ABB RobotStudio station: IRB1600_packaged.rspag

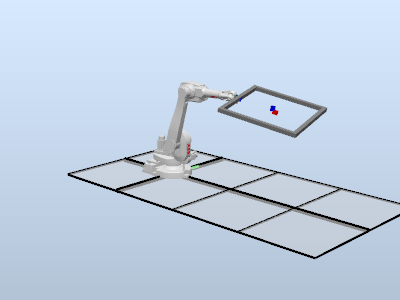
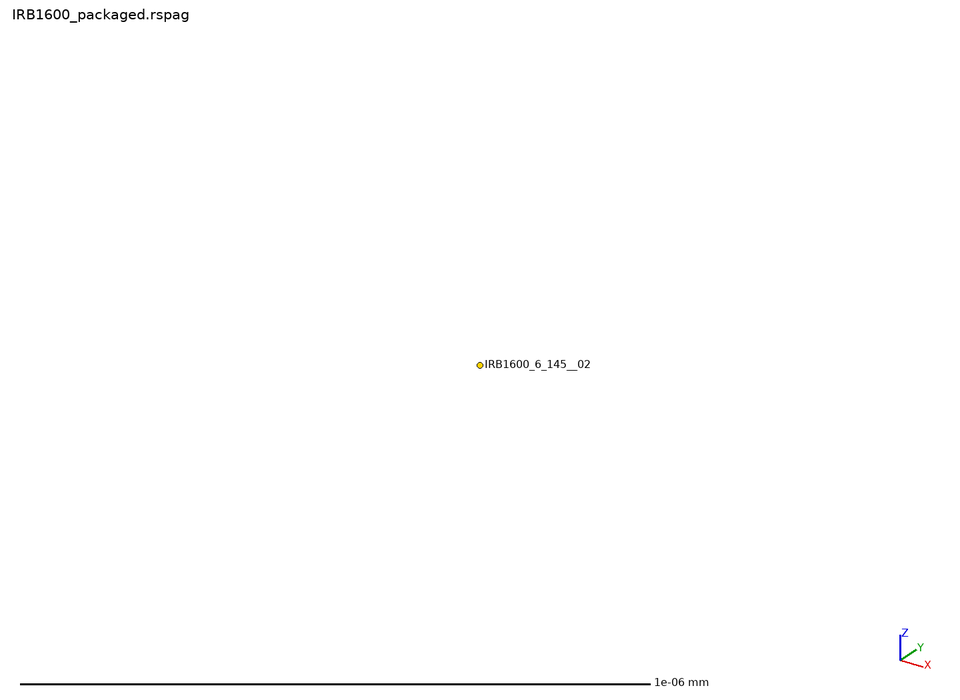
[picture v1: parts stored in the station drawn from their meshes, with robot base, taught points and paths (robot models come from the ABB library and are not in the file)]
--- station ---
Station Solution1 (saved by RobotStudio 22.2.9947.0)
Controller IRB1600_6_145
  mechanical unit ROB_1: IRB1600_6_145__02, 6 joints, base frame (0, 0, 0) mm
Layout (positions relative to the parent item):
  - IRB1600_6_145__02 [mechanism, from Robots\IRB1600_6_145_G_02.rslib] at (0, 0, 0) mm; joint values [0.1292, 0.2457, -0.2431, -2.5339, -0.2406, 2.6375] (rad or m)
  - flange_connector [part, from Tools\IsoPlate_small_Binzel.rslib] at (974.03, 135.42, 1151.03) mm, rotated rx 149.84 ry 76.75 rz 164.54 deg
  - plane [part] at (1455.82, 269.91, 1054.92) mm, rotated rx 173.25 ry -11.43 rz -164.62 deg, size 1000 x 1000 x 50 mm
  - Frame_1 [frame]
  - Frame_2 [frame] at (-23.65, -1.83, 250.36) mm
Attachment: flange_connector is attached to IRB1600_6_145__02 / Link6
Attachment: plane is attached to flange_connector
Attachment: Workobject_2 is attached to IRB1600_6_145__02 / Link1
Targets, tools, work objects and paths stored in the station and not in the controller backup, written as RAPID:
! task T_ROB1
MODULE Module1
  LOCAL PERS wobjdata egm_wobj:=[FALSE,TRUE,"",[[0,0,0],[1,0,0,0]],[[0,0,0],[1,0,0,0]]];
  PROC EGM_CARTESIAN_MOVE()
    WaitTime 2;
  ENDPROC
ENDMODULE


--- Backups/IRB1600_6_145/RAPID/TASK1/PROGMOD/CalibData.mod ---
MODULE CalibData
    TASK PERS tooldata Tooldata_3:=[TRUE,[[-23.481,11.123,47.179],[0.707106781,0,0.707106781,0]],[1,[0,0,1],[1,0,0,0],0,0,0]];
    TASK PERS tooldata Tooldata_8:=[TRUE,[[35.292999999,18.761,1471.373000001],[0.707106781,0,-0.707106781,0]],[1,[0,0,1],[1,0,0,0],0,0,0]];
    TASK PERS tooldata Tooldata_4:=[TRUE,[[0,0,0],[1,0,0,0]],[1,[0,0,1],[1,0,0,0],0,0,0]];
    TASK PERS tooldata Tooldata_5:=[TRUE,[[0,0,0],[1,0,0,0]],[1,[0,0,1],[1,0,0,0],0,0,0]];
    TASK PERS tooldata Tooldata_6:=[TRUE,[[0,0,0],[1,0,0,0]],[1,[0,0,1],[1,0,0,0],0,0,0]];
    TASK PERS tooldata Tooldata_7:=[TRUE,[[-23.772999698,2.161000196,740.120999999],[0.707106781,0,-0.707106781,0]],[1,[0,0,1],[1,0,0,0],0,0,0]];
    TASK PERS wobjdata Workobject_2:=[FALSE,TRUE,"ROB_1",[[-55.133477186,-6.202200727,258.13059393],[1,0,0,0]],[[0,0,0],[1,0,0,0]]];
    TASK PERS tooldata Tooldata_9:=[TRUE,[[20.616002648,0.899999913,497.265999882],[0.707106781,-0.000000002,-0.707106781,0]],[1,[0,0,1],[1,0,0,0],0,0,0]];
    TASK PERS wobjdata Wobj_joint1:=[TRUE,FALSE,"ROB_1",[[639.116,-613.962,-938.233],[1,0,0,0]],[[0,0,0],[1,0,0,0]]];
ENDMODULE

--- Backups/IRB1600_6_145/RAPID/TASK1/PROGMOD/Module1.mod ---
MODULE Module1

     VAR robtarget position;
     VAR robtarget starting_position;
     VAR jointtarget joints;
     VAR speeddata velocity;
    TASK PERS wobjdata wobj:=[FALSE,FALSE,"ROB_1",[[639.116,-22.796,-980.437],[1,0,0,0]],[[0,0,0],[1,0,0,0]]];

    PROC main()

starting_position := CRobT(\TaskName:="T_ROB1" \Tool:=Tooldata_9 \WObj:=Workobject_2);
move 64,-487.9,0,3.2,0,1.3;
move 64,-487.9,0,3.2,15,1.4;
move 64,-487.9,0,3.6,15,1.4;
move 65,-487.9,-0,3.6,15,1.4;
move 65,-487.9,-0,3.6,15,1.5;
move 65,-487.9,-0.1,3.6,15,1.5;
move 65,-487.9,-0.1,3.6,15,1.6;
move 65,-487.9,-0.1,3.6,15,1.6;
move 66,-488,-0.1,3.6,15,1.7;
move 66,-488.1,-0.2,3.6,14.9,1.7;
move 66,-488.1,-0.2,3.6,14.9,1.8;
move 66,-488.2,-0.2,3.6,14.9,1.9;
move 66,-488.3,-0.2,3.6,14.9,1.9;
move 66,-488.5,-0.3,3.6,14.9,2;
move 66,-488.6,-0.3,3.6,14.9,2.1;
move 66,-488.8,-0.3,3.6,14.8,2.1;
move 66,-489,-0.3,3.6,14.8,2.2;
move 66,-489.3,-0.4,3.6,14.8,2.3;
move 66,-489.6,-0.4,3.6,14.8,2.3;
move 66,-489.9,-0.4,3.6,14.8,2.4;
move 66,-490.4,-0.5,3.6,14.7,2.5;
move 66,-490.8,-0.5,3.6,14.7,2.5;
move 66,-491.3,-0.5,3.6,14.7,2.6;
move 66,-491.9,-0.6,3.6,14.6,2.7;
move 66,-492.5,-0.6,3.6,14.6,2.8;
move 66,-493.2,-0.6,3.6,14.6,2.9;
move 65,-493.9,-0.7,3.6,14.5,2.9;
move 65,-494.7,-0.7,3.6,14.5,3;
move 65,-495.5,-0.7,3.6,14.5,3.1;
move 65,-496.4,-0.8,3.6,14.4,3.2;
move 64,-497.4,-0.8,3.6,14.4,3.3;
move 64,-498.4,-0.8,3.6,14.3,3.4;
move 63,-499.4,-0.9,3.6,14.3,3.5;
move 62,-500.5,-0.9,3.2,14.2,3.6;
move 62,-501.6,-0.9,3.2,14.2,3.7;
move 61,-502.7,-1,3.2,14.1,3.8;
move 60,-503.8,-1,3.2,14.1,3.8;
move 60,-504.9,-1,3.2,14,3.9;
move 59,-506,-1.1,3.2,14,4;
move 58,-507.1,-1.1,3.2,13.9,4.1;
move 57,-508.2,-1.1,3.2,13.9,4.2;
move 56,-509.2,-1.2,2.8,13.8,4.3;
move 55,-510.3,-1.2,2.8,13.8,4.4;
move 54,-511.3,-1.2,2.8,13.7,4.5;
move 53,-512.3,-1.3,2.8,13.6,4.6;
move 52,-513.2,-1.3,2.8,13.6,4.7;
move 51,-514,-1.3,2.4,13.5,4.8;
move 50,-514.8,-1.3,2.4,13.5,4.9;
move 49,-515.5,-1.4,2.4,13.4,5;
move 47,-516.2,-1.4,2.4,13.3,5.1;
move 46,-516.8,-1.4,2.4,13.3,5.2;
move 45,-517.3,-1.4,2,13.2,5.3;
move 44,-517.7,-1.4,2,13.1,5.4;
move 42,-518.1,-1.4,2,13,5.5;
move 41,-518.3,-1.5,2,13,5.6;
move 39,-518.5,-1.5,1.6,12.9,5.7;
move 38,-518.6,-1.5,1.6,12.8,5.8;
move 37,-518.6,-1.5,1.6,12.7,5.9;
move 35,-518.5,-1.5,1.6,12.7,6;
move 34,-518.3,-1.5,1.2,12.6,6.1;
move 32,-518.1,-1.5,1.2,12.5,6.2;
move 31,-517.8,-1.5,1.2,12.4,6.2;
move 30,-517.5,-1.6,1.2,12.3,6.3;
move 28,-517.2,-1.6,0.8,12.3,6.4;
move 27,-516.8,-1.6,0.8,12.2,6.5;
move 25,-516.4,-1.6,0.8,12.1,6.6;
move 24,-516.1,-1.6,0.8,12,6.7;
move 22,-515.7,-1.5,0.4,11.9,6.8;
move 21,-515.3,-1.5,0.4,11.8,6.9;
move 20,-515,-1.5,0.4,11.7,7;
move 18,-514.6,-1.5,0.4,11.6,7;
move 17,-514.3,-1.5,0,11.6,7.1;
move 15,-514.1,-1.5,0,11.5,7.2;
move 14,-513.8,-1.5,-0,11.4,7.3;
move 13,-513.7,-1.5,-0,11.3,7.4;
move 12,-513.5,-1.5,-0.4,11.2,7.5;
move 10,-513.4,-1.5,-0.4,11.1,7.5;
move 9,-513.3,-1.4,-0.4,11,7.6;
move 8,-513.2,-1.4,-0.4,10.9,7.7;
move 7,-513.2,-1.4,-0.4,10.8,7.8;
move 6,-513.2,-1.4,-0.8,10.7,7.9;
move 4,-513.2,-1.4,-0.8,10.6,7.9;
move 3,-513.2,-1.3,-0.8,10.5,8;
move 2,-513.1,-1.3,-0.8,10.4,8.1;
move 1,-513.1,-1.3,-0.8,10.3,8.2;
move 0,-513.1,-1.3,-1.2,10.2,8.2;
move -1,-513.1,-1.3,-1.2,10.1,8.3;
move -2,-513,-1.2,-1.2,9.9,8.4;
move -3,-513,-1.2,-1.2,9.8,8.4;
move -4,-512.9,-1.2,-1.2,9.7,8.5;
move -5,-512.8,-1.2,-1.2,9.6,8.6;
move -5,-512.7,-1.2,-1.6,9.5,8.7;
move -6,-512.5,-1.1,-1.6,9.4,8.7;
move -7,-512.3,-1.1,-1.6,9.3,8.8;
move -7,-512,-1.1,-1.6,9.2,8.9;
move -7,-511.7,-1.1,-1.6,9,8.9;
move -8,-511.4,-1,-1.6,8.9,9;
move -8,-511,-1,-1.6,8.8,9.1;
move -8,-510.6,-1,-1.6,8.7,9.1;
move -8,-510.2,-1,-1.6,8.6,9.2;
move -8,-509.7,-1,-1.6,8.5,9.3;
move -8,-509.1,-1,-1.6,8.3,9.3;
move -8,-508.6,-0.9,-1.6,8.2,9.4;
move -8,-508,-0.9,-1.6,8.1,9.4;
move -9,-507.4,-0.9,-1.6,8,9.5;
move -9,-506.8,-0.9,-1.6,7.9,9.6;
move -9,-506.2,-0.9,-1.6,7.7,9.6;
move -9,-505.6,-0.9,-2,7.6,9.7;
move -9,-505,-0.9,-1.6,7.5,9.7;
move -9,-504.4,-0.8,-1.6,7.4,9.8;
move -9,-503.8,-0.8,-1.6,7.2,9.8;
move -8,-503.2,-0.8,-1.6,7.1,9.9;
move -8,-502.7,-0.8,-1.6,7,9.9;
move -8,-502.2,-0.8,-1.6,6.9,10;
move -8,-501.7,-0.8,-1.6,6.7,10;
move -8,-501.2,-0.8,-1.6,6.6,10.1;
move -8,-500.8,-0.8,-1.6,6.5,10.1;
move -7,-500.4,-0.7,-1.6,6.4,10.2;
move -7,-500,-0.7,-1.6,6.2,10.2;
move -7,-499.7,-0.7,-1.6,6.1,10.3;
move -6,-499.4,-0.7,-1.6,6,10.3;
move -6,-499.1,-0.7,-1.6,5.8,10.4;
move -5,-498.8,-0.7,-1.2,5.7,10.4;
move -4,-498.6,-0.7,-1.2,5.6,10.4;
move -4,-498.3,-0.7,-1.2,5.5,10.5;
move -3,-498.1,-0.7,-1.2,5.3,10.5;
move -2,-497.9,-0.7,-1.2,5.2,10.5;
move -1,-497.7,-0.7,-1.2,5.1,10.6;
move -1,-497.5,-0.6,-1.2,4.9,10.6;
move 0,-497.3,-0.6,-1.2,4.8,10.6;
move 1,-497.1,-0.6,-0.8,4.7,10.7;
move 2,-496.9,-0.6,-0.8,4.5,10.7;
move 3,-496.8,-0.6,-0.8,4.4,10.7;
move 4,-496.6,-0.6,-0.8,4.3,10.7;
move 5,-496.5,-0.6,-0.8,4.1,10.8;
move 6,-496.4,-0.6,-0.8,4,10.8;
move 7,-496.3,-0.6,-0.4,3.9,10.8;
move 7,-496.1,-0.6,-0.4,3.7,10.8;
move 8,-496,-0.6,-0.4,3.6,10.8;
move 9,-495.9,-0.6,-0.4,3.5,10.9;
move 10,-495.8,-0.6,-0.4,3.3,10.9;
move 11,-495.8,-0.6,-0.4,3.2,10.9;
move 12,-495.7,-0.6,-0,3,10.9;
move 12,-495.6,-0.5,-0,2.9,10.9;
move 13,-495.6,-0.5,-0,2.8,10.9;
move 14,-495.5,-0.5,-0,2.6,10.9;
move 14,-495.5,-0.5,0,2.5,10.9;
move 14,-495.5,-0.5,0,2.4,10.9;
move 15,-495.6,-0.5,0,2.2,11;
move 15,-495.6,-0.5,0,2.1,11;
move 16,-495.7,-0.5,0,2,11;
move 16,-495.8,-0.5,0,1.8,11;
move 17,-495.9,-0.5,0,1.7,11;
move 17,-496,-0.5,0,1.6,11;
move 18,-496.2,-0.5,0.4,1.4,11;
move 18,-496.4,-0.5,0.4,1.3,11;
move 19,-496.6,-0.4,0.4,1.1,11;
move 19,-496.8,-0.4,0.4,1,11;
move 20,-497.1,-0.4,0.4,0.9,11;
move 20,-497.4,-0.4,0.4,0.7,11;
move 20,-497.8,-0.4,0.4,0.6,11;
move 20,-498.2,-0.4,0.4,0.5,11;
move 20,-498.6,-0.4,0.4,0.3,11;
move 19,-499.1,-0.4,0.4,0.2,11;
move 19,-499.6,-0.4,0.4,0.1,11;
move 18,-500.1,-0.4,0.4,-0.1,11;
move 18,-500.7,-0.4,0.4,-0.2,11;
move 17,-501.2,-0.4,0,-0.3,11;
move 16,-501.8,-0.4,0,-0.5,11;
move 16,-502.4,-0.3,0,-0.6,11;
move 15,-503,-0.3,0,-0.7,11;
move 15,-503.6,-0.3,0,-0.9,11;
move 14,-504.3,-0.3,-0,-1,11;
move 13,-504.8,-0.3,-0,-1.1,11;
move 13,-505.4,-0.3,-0,-1.3,11;
move 12,-506,-0.3,-0,-1.4,11;
move 11,-506.5,-0.3,-0.4,-1.5,11;
move 10,-506.9,-0.3,-0.4,-1.7,11;
move 9,-507.3,-0.3,-0.4,-1.8,11;
move 8,-507.7,-0.3,-0.4,-1.9,11;
move 7,-508,-0.3,-0.4,-2,11;
move 6,-508.3,-0.3,-0.4,-2.2,11;
move 5,-508.5,-0.3,-0.8,-2.3,11;
move 4,-508.6,-0.3,-0.8,-2.4,11;
move 3,-508.7,-0.3,-0.8,-2.6,11;
move 2,-508.8,-0.3,-0.8,-2.7,11;
move 1,-508.7,-0.3,-0.8,-2.8,10.9;
move -1,-508.6,-0.3,-1.2,-2.9,10.9;
move -2,-508.5,-0.3,-1.2,-3.1,10.9;
move -3,-508.3,-0.2,-1.2,-3.2,10.9;
move -5,-508,-0.2,-1.2,-3.3,10.9;
move -6,-507.7,-0.2,-1.6,-3.4,10.9;
move -7,-507.3,-0.2,-1.6,-3.6,10.9;
move -9,-506.9,-0.2,-1.6,-3.7,10.9;
move -10,-506.5,-0.2,-1.6,-3.8,10.8;
move -11,-506,-0.2,-2,-3.9,10.8;
move -12,-505.4,-0.2,-2,-4,10.8;
move -14,-504.9,-0.2,-2,-4.2,10.8;
move -15,-504.3,-0.2,-2,-4.3,10.8;
move -16,-503.7,-0.2,-2,-4.4,10.7;
move -17,-503.1,-0.2,-2.4,-4.5,10.7;
move -18,-502.5,-0.2,-2.4,-4.6,10.7;
move -19,-501.8,-0.1,-2.4,-4.8,10.7;
move -20,-501.2,-0.1,-2.4,-4.9,10.6;
move -21,-500.6,-0.1,-2.4,-5,10.6;
move -22,-500,-0.1,-2.8,-5.1,10.6;
move -23,-499.4,-0.1,-2.8,-5.2,10.6;
move -24,-498.8,-0.1,-2.8,-5.3,10.5;
move -25,-498.2,-0.1,-2.8,-5.5,10.5;
move -26,-497.6,-0.1,-2.8,-5.6,10.5;
move -27,-497.1,-0,-2.8,-5.7,10.4;
move -27,-496.6,0,-2.8,-5.8,10.4;
move -28,-496,0,-3.2,-5.9,10.3;
move -29,-495.5,0,-3.2,-6,10.3;
move -30,-495,0,-3.2,-6.1,10.3;
move -30,-494.5,0.1,-3.2,-6.2,10.2;
move -31,-493.9,0.1,-3.2,-6.3,10.2;
move -31,-493.4,0.1,-3.2,-6.4,10.1;
move -32,-492.8,0.2,-3.2,-6.5,10.1;
move -32,-492.2,0.2,-3.2,-6.6,10;
move -32,-491.7,0.2,-3.6,-6.7,10;
move -33,-491.1,0.3,-3.2,-6.9,9.9;
move -33,-490.4,0.3,-3.2,-7,9.9;
move -33,-489.8,0.3,-3.2,-7.1,9.8;
move -33,-489.2,0.3,-3.6,-7.2,9.8;
move -33,-488.5,0.4,-3.6,-7.3,9.7;
move -33,-487.9,0.4,-3.6,-7.4,9.7;
move -33,-487.3,0.4,-3.6,-7.4,9.6;
move -33,-486.7,0.5,-3.2,-7.5,9.6;
move -32,-486.1,0.5,-3.2,-7.6,9.5;
move -32,-485.5,0.6,-3.2,-7.7,9.5;
move -32,-485,0.6,-3.2,-7.8,9.4;
move -31,-484.4,0.6,-3.2,-7.9,9.4;
move -31,-483.9,0.7,-3.2,-8,9.3;
move -31,-483.4,0.7,-3.2,-8.1,9.2;
move -31,-482.9,0.8,-3.2,-8.2,9.2;
move -30,-482.5,0.8,-3.2,-8.3,9.1;
move -30,-482,0.9,-3.2,-8.4,9.1;
move -29,-481.6,0.9,-3.2,-8.5,9;
move -29,-481.2,0.9,-3.2,-8.5,9;
move -28,-480.8,1,-3.2,-8.6,8.9;
move -27,-480.4,1,-2.8,-8.7,8.8;
move -26,-480,1.1,-2.8,-8.8,8.8;
move -26,-479.5,1.1,-2.8,-8.9,8.7;
move -25,-479.1,1.2,-2.8,-9,8.6;
move -24,-478.6,1.2,-2.8,-9,8.6;
move -23,-478.1,1.3,-2.8,-9.1,8.5;
move -22,-477.6,1.3,-2.4,-9.2,8.5;
move -20,-477.1,1.4,-2.4,-9.3,8.4;
move -19,-476.5,1.4,-2.4,-9.4,8.3;
move -18,-475.9,1.5,-2.4,-9.4,8.3;
move -17,-475.3,1.5,-2.4,-9.5,8.2;
move -16,-474.7,1.6,-2,-9.6,8.1;
move -14,-474.1,1.6,-2,-9.7,8.1;
move -13,-473.4,1.7,-2,-9.7,8;
move -12,-472.7,1.7,-2,-9.8,7.9;
move -10,-472,1.7,-1.6,-9.9,7.9;
move -9,-471.4,1.8,-1.6,-9.9,7.8;
move -8,-470.7,1.8,-1.6,-10,7.7;
move -6,-470,1.9,-1.6,-10.1,7.7;
move -5,-469.4,1.9,-1.2,-10.1,7.6;
move -4,-468.8,1.9,-1.2,-10.2,7.5;
move -3,-468.3,2,-1.2,-10.3,7.4;
move -1,-467.9,2,-1.2,-10.3,7.4;
move 0,-467.5,2.1,-1.2,-10.4,7.3;
move 1,-467.2,2.1,-0.8,-10.4,7.2;
move 3,-467,2.1,-0.8,-10.5,7.1;
move 4,-466.9,2.1,-0.8,-10.5,7.1;
move 5,-466.9,2.2,-0.8,-10.6,7;
move 7,-466.9,2.2,-0.4,-10.7,6.9;
move 8,-467,2.2,-0.4,-10.7,6.9;
move 10,-467.2,2.2,-0.4,-10.8,6.8;
move 11,-467.5,2.3,-0.4,-10.8,6.7;
move 12,-467.9,2.3,-0,-10.9,6.6;
move 14,-468.3,2.3,-0,-10.9,6.5;
move 15,-468.8,2.3,0,-11,6.5;
move 16,-469.4,2.3,0,-11,6.4;
move 17,-470,2.3,0.4,-11.1,6.3;
move 18,-470.7,2.3,0.4,-11.1,6.2;
move 20,-471.4,2.3,0.4,-11.1,6.2;
move 21,-472.1,2.3,0.4,-11.2,6.1;
move 21,-472.8,2.3,0.4,-11.2,6;
move 22,-473.6,2.3,0.4,-11.3,5.9;
move 23,-474.3,2.3,0.8,-11.3,5.8;
move 24,-475.1,2.3,0.8,-11.4,5.8;
move 25,-475.8,2.3,0.8,-11.4,5.7;
move 25,-476.5,2.3,0.8,-11.4,5.6;
move 26,-477.1,2.3,0.8,-11.5,5.5;
move 26,-477.8,2.3,0.8,-11.5,5.4;
move 27,-478.3,2.3,0.8,-11.5,5.4;
move 27,-478.9,2.2,0.8,-11.6,5.3;
move 28,-479.4,2.2,0.8,-11.6,5.2;
move 28,-479.8,2.2,0.8,-11.6,5.1;
move 29,-480.2,2.2,1.2,-11.7,5;
move 30,-480.6,2.1,1.2,-11.7,5;
move 30,-480.9,2.1,1.2,-11.7,4.9;
move 31,-481.2,2.1,1.2,-11.7,4.8;
move 31,-481.5,2.1,1.2,-11.8,4.7;
move 31,-481.7,2,1.2,-11.8,4.6;
move 31,-481.9,2,1.2,-11.8,4.5;
move 31,-482.1,2,1.2,-11.8,4.5;
move 32,-482.2,1.9,1.2,-11.8,4.4;
move 32,-482.4,1.9,1.2,-11.9,4.3;
move 32,-482.5,1.8,1.2,-11.9,4.2;
move 32,-482.6,1.8,1.2,-11.9,4.1;
move 32,-482.7,1.8,1.2,-11.9,4;
move 32,-482.8,1.7,1.2,-11.9,4;
move 32,-482.9,1.7,1.2,-11.9,3.9;
move 32,-483,1.6,1.2,-12,3.8;
move 32,-483.1,1.6,1.2,-12,3.7;
move 32,-483.2,1.5,1.2,-12,3.6;
move 32,-483.2,1.5,1.2,-12,3.5;
move 32,-483.2,1.4,1.2,-12,3.5;
move 32,-483.3,1.4,1.2,-12,3.4;
move 31,-483.3,1.3,1.2,-12,3.3;
move 31,-483.3,1.3,1.2,-12,3.2;
move 31,-483.3,1.2,1.2,-12,3.1;
move 31,-483.3,1.2,1.2,-12,3;
move 30,-483.4,1.1,1.2,-12,2.9;
move 30,-483.4,1.1,1.2,-12,2.9;
move 29,-483.4,1,1.2,-12,2.8;
move 29,-483.5,1,0.8,-12,2.7;
move 28,-483.5,0.9,0.8,-12,2.6;
move 27,-483.5,0.9,0.8,-12,2.5;
move 27,-483.5,0.8,0.8,-12,2.4;
move 27,-483.5,0.8,0.8,-12,2.3;
move 26,-483.5,0.8,0.8,-12,2.3;
move 26,-483.5,0.7,0.8,-12,2.2;
move 26,-483.5,0.7,0.8,-12,2.1;
move 26,-483.5,0.6,0.8,-12,2;
move 26,-483.5,0.6,0.8,-12,1.9;
move 26,-483.5,0.5,0.8,-12,1.8;
move 26,-483.5,0.4,0.8,-12,1.7;
move 26,-483.5,0.4,0.8,-11.9,1.7;
move 26,-483.5,0.3,0.8,-11.9,1.6;
move 27,-483.5,0.3,0.8,-11.9,1.5;
move 27,-483.5,0.3,0.8,-11.9,1.4;
move 27,-483.5,0.2,0.8,-11.9,1.3;
move 28,-483.5,0.1,0.8,-11.9,1.2;
move 28,-483.5,0.1,0.8,-11.9,1.2;
move 29,-483.5,0,1.2,-11.8,1.1;
move 30,-483.5,-0,1.2,-11.8,1;
move 30,-483.5,-0.1,1.2,-11.8,0.9;
move 31,-483.5,-0.1,1.2,-11.8,0.8;
move 31,-483.5,-0.1,1.2,-11.8,0.7;
move 31,-483.5,-0.1,1.2,-11.7,0.7;
move 31,-483.5,-0.2,1.2,-11.7,0.6;
move 31,-483.5,-0.3,1.2,-11.7,0.5;
move 32,-483.5,-0.3,1.2,-11.7,0.4;
move 32,-483.5,-0.3,1.2,-11.6,0.3;
move 32,-483.5,-0.4,1.2,-11.6,0.2;
move 32,-483.5,-0.4,1.2,-11.6,0.2;
move 32,-483.5,-0.5,1.2,-11.5,0.1;
move 33,-483.5,-0.5,1.2,-11.5,-0;
move 33,-483.5,-0.5,1.2,-11.5,-0.1;
move 34,-483.5,-0.6,1.2,-11.5,-0.2;
move 34,-483.5,-0.6,1.2,-11.4,-0.3;
move 35,-483.5,-0.7,1.6,-11.4,-0.3;
move 35,-483.5,-0.7,1.6,-11.4,-0.4;
move 36,-483.5,-0.7,1.6,-11.3,-0.5;
move 36,-483.5,-0.8,1.6,-11.3,-0.6;
move 37,-483.5,-0.8,1.6,-11.3,-0.7;
move 37,-483.5,-0.9,1.6,-11.2,-0.7;
move 38,-483.5,-0.9,1.6,-11.2,-0.8;
move 38,-483.6,-1,1.6,-11.1,-0.9;
move 39,-483.6,-1,1.6,-11.1,-1;
move 39,-483.7,-1,1.6,-11.1,-1;
move 40,-483.7,-1.1,1.6,-11,-1.1;
move 40,-483.9,-1.1,2,-11,-1.2;
move 41,-484,-1.2,2,-10.9,-1.3;
move 41,-484.2,-1.2,2,-10.9,-1.4;
move 41,-484.3,-1.2,2,-10.9,-1.4;
move 42,-484.5,-1.2,1.6,-10.8,-1.5;
move 42,-484.8,-1.3,2,-10.8,-1.6;
move 42,-485,-1.3,2,-10.7,-1.7;
move 42,-485.3,-1.3,2,-10.7,-1.7;
move 43,-485.7,-1.3,2,-10.6,-1.8;
move 43,-486,-1.4,2,-10.6,-1.9;
move 43,-486.4,-1.4,2,-10.5,-2;
move 43,-486.8,-1.4,2,-10.5,-2;
move 43,-487.3,-1.4,2,-10.4,-2.1;
move 43,-487.8,-1.4,2,-10.4,-2.2;
move 42,-488.3,-1.5,2,-10.4,-2.3;
move 42,-488.8,-1.5,2,-10.3,-2.3;
move 42,-489.4,-1.5,2,-10.3,-2.4;
move 41,-490,-1.5,2,-10.2,-2.5;
move 40,-490.7,-1.5,2,-10.1,-2.5;
move 40,-491.3,-1.5,1.6,-10.1,-2.6;
move 39,-491.9,-1.5,1.6,-10,-2.7;
move 38,-492.6,-1.5,1.6,-10,-2.8;
move 38,-493.2,-1.5,1.6,-9.9,-2.8;
move 37,-493.9,-1.6,1.6,-9.9,-2.9;
move 36,-494.5,-1.6,1.6,-9.8,-3;
move 35,-495.2,-1.5,1.6,-9.8,-3;
move 34,-495.9,-1.5,1.6,-9.7,-3.1;
move 34,-496.5,-1.5,1.2,-9.7,-3.2;
move 33,-497.2,-1.5,1.2,-9.6,-3.2;
move 31,-497.9,-1.5,1.2,-9.6,-3.3;
move 30,-498.6,-1.5,1.2,-9.5,-3.4;
move 29,-499.3,-1.5,1.2,-9.4,-3.4;
move 27,-500,-1.5,0.8,-9.4,-3.5;
move 26,-500.7,-1.5,0.8,-9.3,-3.6;
move 24,-501.5,-1.4,0.8,-9.3,-3.6;
move 23,-502.2,-1.4,0.8,-9.2,-3.7;
move 21,-503,-1.3,0.4,-9.1,-3.7;
move 19,-503.7,-1.3,0.4,-9.1,-3.8;
move 17,-504.5,-1.3,0,-9,-3.9;
move 15,-505.2,-1.2,0,-9,-3.9;
move 13,-505.9,-1.2,-0,-8.9,-4;
move 11,-506.6,-1.1,-0.4,-8.8,-4.1;
move 9,-507.2,-1.1,-0.4,-8.8,-4.1;
move 7,-507.8,-1.1,-0.4,-8.7,-4.2;
move 5,-508.3,-1,-0.8,-8.7,-4.2;
move 3,-508.7,-1,-0.8,-8.6,-4.3;
move 1,-509.1,-0.9,-0.8,-8.5,-4.4;
move -1,-509.3,-0.9,-1.2,-8.5,-4.4;
move -3,-509.5,-0.8,-1.2,-8.4,-4.5;
move -5,-509.6,-0.8,-1.2,-8.3,-4.5;
move -7,-509.6,-0.7,-1.6,-8.3,-4.6;
move -9,-509.6,-0.6,-1.6,-8.2,-4.7;
move -12,-509.4,-0.6,-2,-8.1,-4.7;
move -14,-509.1,-0.5,-2,-8.1,-4.8;
move -16,-508.8,-0.5,-2,-8,-4.8;
move -18,-508.4,-0.4,-2.4,-8,-4.9;
move -21,-507.8,-0.3,-2.4,-7.9,-4.9;
move -23,-507.2,-0.3,-2.8,-7.8,-5;
move -25,-506.6,-0.2,-2.8,-7.8,-5;
move -27,-505.8,-0.1,-2.8,-7.7,-5.1;
move -30,-505.1,-0.1,-3.2,-7.6,-5.2;
move -32,-504.2,-0,-3.2,-7.6,-5.2;
move -34,-503.4,0,-3.6,-7.5,-5.3;
move -36,-502.5,0.1,-3.6,-7.4,-5.3;
move -38,-501.6,0.2,-3.6,-7.4,-5.4;
move -40,-500.6,0.2,-4,-7.3,-5.4;
move -42,-499.6,0.3,-4,-7.2,-5.5;
move -44,-498.6,0.4,-4,-7.2,-5.5;
move -46,-497.7,0.4,-4.4,-7.1,-5.6;
move -48,-496.7,0.5,-4.4,-7,-5.6;
move -50,-495.7,0.6,-4.8,-7,-5.7;
move -52,-494.7,0.6,-4.8,-6.9,-5.7;
move -54,-493.7,0.7,-4.8,-6.8,-5.8;
move -56,-492.6,0.7,-4.8,-6.7,-5.8;
move -57,-491.6,0.8,-5.2,-6.7,-5.9;
move -59,-490.6,0.9,-5.2,-6.6,-5.9;
move -61,-489.6,0.9,-5.2,-6.5,-5.9;
move -62,-488.5,1,-5.6,-6.5,-6;
move -64,-487.5,1,-5.6,-6.4,-6;
move -65,-486.5,1.1,-5.6,-6.3,-6.1;
move -67,-485.4,1.1,-5.6,-6.3,-6.1;
move -68,-484.4,1.2,-6,-6.2,-6.2;
move -69,-483.4,1.2,-6,-6.1,-6.2;
move -70,-482.3,1.3,-6,-6.1,-6.3;
move -72,-481.3,1.3,-6,-6,-6.3;
move -73,-480.3,1.3,-6,-5.9,-6.3;
move -74,-479.2,1.4,-6.4,-5.9,-6.4;
move -75,-478.2,1.4,-6.4,-5.8,-6.4;
move -76,-477.2,1.5,-6.4,-5.7,-6.5;
move -77,-476.2,1.5,-6.4,-5.7,-6.5;
move -78,-475.2,1.5,-6.4,-5.6,-6.5;
move -79,-474.2,1.5,-6.4,-5.5,-6.6;
move -79,-473.2,1.6,-6.8,-5.4,-6.6;
move -80,-472.2,1.6,-6.8,-5.4,-6.6;
move -81,-471.2,1.6,-6.8,-5.3,-6.7;
move -82,-470.2,1.6,-6.8,-5.2,-6.7;
move -83,-469.3,1.7,-6.8,-5.2,-6.8;
move -84,-468.3,1.7,-6.8,-5.1,-6.8;
move -84,-467.3,1.7,-6.8,-5,-6.8;
move -85,-466.4,1.7,-7.2,-5,-6.9;
move -86,-465.4,1.7,-7.2,-4.9,-6.9;
move -86,-464.4,1.7,-7.2,-4.8,-6.9;
move -87,-463.4,1.7,-7.2,-4.8,-7;
move -87,-462.4,1.7,-7.2,-4.7,-7;
move -87,-461.5,1.7,-7.2,-4.6,-7;
move -88,-460.5,1.7,-7.2,-4.6,-7.1;
move -88,-459.5,1.6,-7.2,-4.5,-7.1;
move -88,-458.5,1.6,-7.2,-4.4,-7.1;
move -89,-457.5,1.6,-7.2,-4.4,-7.2;
move -89,-456.5,1.6,-7.2,-4.3,-7.2;
move -90,-455.5,1.6,-7.2,-4.2,-7.2;
move -90,-454.6,1.6,-7.2,-4.2,-7.3;
move -91,-453.6,1.5,-7.6,-4.1,-7.3;
move -91,-452.6,1.5,-7.6,-4,-7.3;
move -92,-451.7,1.5,-7.6,-4,-7.3;
move -92,-450.8,1.5,-7.6,-3.9,-7.4;
move -93,-449.9,1.4,-7.6,-3.8,-7.4;
move -93,-449.1,1.4,-7.6,-3.8,-7.4;
move -93,-448.2,1.4,-7.6,-3.7,-7.5;
move -93,-447.5,1.3,-7.6,-3.6,-7.5;
move -93,-446.8,1.3,-7.6,-3.6,-7.5;
move -94,-446.1,1.2,-7.6,-3.5,-7.5;
move -94,-445.5,1.2,-7.6,-3.4,-7.6;
move -94,-444.9,1.1,-7.6,-3.4,-7.6;
move -94,-444.3,1.1,-7.6,-3.3,-7.6;
move -95,-443.7,1.1,-7.6,-3.2,-7.7;
move -95,-443.2,1,-7.6,-3.2,-7.7;
move -96,-442.7,0.9,-7.6,-3.1,-7.7;
move -97,-442.2,0.9,-8,-3,-7.7;
move -97,-441.7,0.8,-8,-3,-7.7;
move -98,-441.2,0.8,-8,-2.9,-7.8;
move -98,-440.6,0.7,-8,-2.8,-7.8;
move -99,-440,0.7,-8,-2.8,-7.8;
move -100,-439.4,0.6,-8,-2.7,-7.8;
move -100,-438.8,0.5,-8,-2.7,-7.8;
move -101,-438.1,0.5,-8,-2.6,-7.9;
move -102,-437.4,0.4,-8,-2.5,-7.9;
move -102,-436.7,0.4,-8.4,-2.5,-7.9;
move -103,-435.9,0.3,-8.4,-2.4,-7.9;
move -103,-435,0.3,-8.4,-2.3,-7.9;
move -104,-434.2,0.2,-8.4,-2.3,-7.9;
move -105,-433.2,0.1,-8.4,-2.2,-7.9;
move -105,-432.3,0.1,-8.4,-2.2,-7.9;
move -106,-431.2,0,-8.4,-2.1,-7.9;
move -107,-430.1,-0,-8.4,-2,-7.9;
move -107,-429,-0.1,-8.4,-2,-8;
move -108,-427.8,-0.2,-8.8,-1.9,-8;
move -109,-426.6,-0.2,-8.8,-1.8,-8;
move -109,-425.3,-0.3,-8.8,-1.8,-8;
move -110,-424.1,-0.3,-8.8,-1.7,-8;
move -110,-422.8,-0.4,-8.8,-1.7,-8;
move -111,-421.5,-0.4,-8.8,-1.6,-8;
move -112,-420.1,-0.5,-8.8,-1.5,-8;
move -112,-418.8,-0.5,-8.8,-1.5,-8;
move -113,-417.5,-0.6,-8.8,-1.4,-8;
move -114,-416.1,-0.7,-9.2,-1.4,-8;
move -115,-414.7,-0.7,-9.2,-1.3,-8;
move -116,-413.3,-0.7,-9.2,-1.3,-8;
move -116,-411.9,-0.8,-9.2,-1.2,-8;
move -117,-410.5,-0.8,-9.2,-1.1,-8;
move -118,-409.1,-0.8,-9.2,-1.1,-8;
move -119,-407.6,-0.9,-9.6,-1,-8;
move -120,-406.2,-0.9,-9.6,-1,-8;
move -120,-404.8,-0.9,-9.6,-0.9,-8;
move -121,-403.3,-0.9,-9.6,-0.8,-8;
move -121,-401.9,-1,-9.6,-0.8,-8;
move -122,-400.4,-1,-9.6,-0.7,-8;
move -122,-399,-1,-9.6,-0.7,-8;
move -122,-397.5,-1,-9.6,-0.6,-8;
move -123,-396.1,-1,-9.6,-0.6,-8;
move -123,-394.6,-1.1,-9.6,-0.5,-8;
move -124,-393.1,-1.1,-9.6,-0.5,-8;
move -124,-391.7,-1.1,-9.6,-0.4,-8;
move -125,-390.3,-1,-10,-0.3,-8;
move -126,-388.8,-1,-10,-0.3,-8;
move -126,-387.4,-1,-10,-0.2,-8;
move -127,-386,-1,-10,-0.2,-8;
move -128,-384.7,-1,-10,-0.1,-8;
move -128,-383.4,-1,-10,-0.1,-8;
move -129,-382.1,-1,-10,-0,-8;
move -130,-380.9,-0.9,-10,0,-8;
move -130,-379.8,-0.9,-10.4,0.1,-8;
move -131,-378.7,-0.9,-10.4,0.1,-8;
move -132,-377.6,-0.9,-10.4,0.2,-8;
move -132,-376.6,-0.9,-10.4,0.2,-8;
move -133,-375.6,-0.8,-10.4,0.3,-8;
move -133,-374.7,-0.8,-10.4,0.3,-8;
move -134,-373.8,-0.8,-10.4,0.4,-8;
move -134,-372.9,-0.7,-10.4,0.4,-8;
move -135,-372.1,-0.6,-10.4,0.5,-8;
move -135,-371.3,-0.6,-10.4,0.5,-8;
move -136,-370.5,-0.5,-10.4,0.6,-8;
move -136,-369.7,-0.5,-10.8,0.7,-8;
move -137,-368.9,-0.4,-10.8,0.7,-8;
move -138,-368.1,-0.4,-10.8,0.8,-8;
move -138,-367.3,-0.3,-10.8,0.8,-8;
move -139,-366.5,-0.2,-10.8,0.9,-8;
move -140,-365.6,-0.1,-10.8,0.9,-8;
move -141,-364.6,-0.1,-10.8,1,-8;
move -141,-363.6,0,-10.8,1,-8;
move -142,-362.5,0.1,-11.2,1,-8;
move -142,-361.3,0.2,-11.2,1.1,-8;
move -143,-360.1,0.3,-11.2,1.1,-8;
move -144,-358.7,0.4,-11.2,1.2,-8;
move -144,-357.4,0.4,-11.2,1.2,-8;
move -144,-355.9,0.5,-11.2,1.3,-8;
move -145,-354.4,0.6,-11.2,1.3,-8;
move -145,-352.8,0.7,-11.2,1.4,-8;
move -146,-351.2,0.8,-11.2,1.4,-8;
move -146,-349.5,0.9,-11.2,1.5,-8;
move -147,-347.7,1,-11.2,1.5,-8;
move -148,-345.9,1.1,-11.6,1.6,-8;
move -148,-344.1,1.2,-11.6,1.6,-8;
move -149,-342.3,1.3,-11.6,1.7,-7.9;
move -149,-340.4,1.4,-11.6,1.7,-7.9;
move -150,-338.5,1.6,-11.6,1.8,-7.9;
move -150,-336.7,1.7,-11.6,1.8,-7.9;
move -150,-334.8,1.8,-11.6,1.9,-7.9;
move -150,-332.9,1.9,-11.6,1.9,-7.9;
move -151,-331.1,2,-11.6,1.9,-7.9;
move -151,-329.3,2.1,-11.6,2,-7.9;
move -152,-327.5,2.2,-11.6,2,-7.9;
move -152,-325.7,2.3,-11.6,2.1,-7.8;
move -153,-323.9,2.4,-11.6,2.1,-7.8;
move -153,-322.2,2.6,-12,2.2,-7.8;
move -154,-320.5,2.7,-12,2.2,-7.8;
move -154,-318.8,2.8,-12,2.3,-7.8;
move -155,-317.1,2.9,-12,2.3,-7.7;
move -155,-315.5,3,-12,2.3,-7.7;
move -155,-313.9,3.2,-12,2.4,-7.7;
move -156,-312.3,3.3,-12,2.4,-7.7;
move -156,-310.8,3.4,-12,2.5,-7.7;
move -156,-309.3,3.5,-12,2.5,-7.6;
move -156,-307.8,3.7,-12,2.6,-7.6;
move -156,-306.4,3.8,-12,2.6,-7.6;
move -156,-305.1,3.9,-12,2.6,-7.6;
move -156,-303.7,4,-12,2.7,-7.5;
move -156,-302.4,4.2,-12,2.7,-7.5;
move -156,-301.1,4.3,-12,2.8,-7.5;
move -156,-299.8,4.4,-12,2.8,-7.5;
move -156,-298.6,4.5,-12,2.9,-7.4;
move -156,-297.3,4.7,-12,2.9,-7.4;
move -156,-296,4.8,-12,2.9,-7.4;
move -156,-294.7,4.9,-12,3,-7.3;
move -156,-293.5,5,-12,3,-7.3;
move -156,-292.2,5.2,-12,3.1,-7.3;
move -156,-290.9,5.3,-12,3.1,-7.3;
move -156,-289.7,5.4,-12,3.2,-7.2;
move -156,-288.4,5.5,-12,3.2,-7.2;
move -156,-287,5.6,-12,3.2,-7.2;
move -156,-285.7,5.8,-12,3.3,-7.2;
move -156,-284.3,5.9,-12,3.3,-7.1;
move -156,-282.9,6,-12,3.4,-7.1;
move -156,-281.5,6.1,-12,3.4,-7.1;
move -156,-280,6.2,-12,3.4,-7.1;
move -156,-278.5,6.3,-12,3.5,-7;
move -156,-277,6.4,-12,3.5,-7;
move -156,-275.5,6.5,-12,3.6,-7;
move -156,-274,6.6,-12,3.6,-6.9;
move -156,-272.4,6.7,-12,3.7,-6.9;
move -156,-270.7,6.8,-12,3.7,-6.9;
move -156,-269.1,6.9,-12,3.7,-6.9;
move -156,-267.4,7,-12,3.8,-6.8;
move -156,-265.6,7.1,-12,3.8,-6.8;
move -156,-263.8,7.2,-12,3.9,-6.8;
move -156,-262,7.3,-12,3.9,-6.8;
move -156,-260.2,7.4,-12,3.9,-6.7;
move -156,-258.3,7.5,-12,4,-6.7;
move -156,-256.4,7.6,-12,4,-6.7;
move -156,-254.5,7.7,-12,4.1,-6.6;
move -156,-252.6,7.7,-12,4.1,-6.6;
move -156,-250.8,7.8,-12,4.1,-6.6;
move -156,-248.9,7.9,-12,4.2,-6.5;
move -156,-247,8,-12,4.2,-6.5;
move -156,-245.2,8.1,-12,4.3,-6.5;
move -156,-243.4,8.1,-12,4.3,-6.4;
move -156,-241.6,8.2,-12,4.3,-6.4;
move -156,-239.9,8.3,-12,4.4,-6.4;
move -156,-238.1,8.3,-12,4.4,-6.3;
move -156,-236.4,8.4,-12,4.5,-6.3;
move -156,-234.7,8.5,-12,4.5,-6.3;
move -156,-233.1,8.5,-12,4.5,-6.2;
move -156,-231.5,8.6,-12,4.6,-6.2;
move -156,-229.9,8.6,-12,4.6,-6.2;
move -156,-228.3,8.7,-12,4.6,-6.1;
move -156,-226.7,8.8,-12,4.7,-6.1;
move -156,-225.2,8.8,-12,4.7,-6.1;
move -156,-223.7,8.8,-12,4.8,-6;
move -156,-222.1,8.9,-12,4.8,-6;
move -156,-220.6,8.9,-12,4.8,-6;
move -156,-219.2,9,-12,4.9,-5.9;
move -156,-217.7,9,-12,4.9,-5.9;
move -156,-216.3,9,-12,5,-5.8;
move -156,-214.9,9.1,-12,5,-5.8;
move -156,-213.5,9.1,-12,5,-5.8;
move -156,-212.2,9.1,-12,5.1,-5.7;
move -156,-210.9,9.1,-12,5.1,-5.7;
move -156,-209.6,9.1,-12,5.2,-5.7;
move -157,-208.4,9.1,-12,5.2,-5.6;
move -157,-207.1,9.1,-12,5.2,-5.6;
move -157,-205.8,9.1,-12,5.3,-5.5;
move -158,-204.5,9.1,-12,5.3,-5.5;
move -158,-203.2,9.1,-12,5.3,-5.5;
move -159,-201.9,9.1,-12.4,5.4,-5.4;
move -160,-200.6,9.1,-12.4,5.4,-5.4;
move -160,-199.3,9.1,-12.4,5.5,-5.3;
move -160,-198,9.1,-12.4,5.5,-5.3;
move -161,-196.7,9.1,-12.4,5.5,-5.2;
move -161,-195.3,9,-12.4,5.6,-5.2;
move -162,-194,9,-12.4,5.6,-5.2;
move -162,-192.7,9,-12.4,5.7,-5.1;
move -162,-191.2,8.9,-12.4,5.7,-5.1;
move -163,-189.8,8.9,-12.4,5.7,-5;
move -163,-188.2,8.9,-12.4,5.8,-5;
move -164,-186.7,8.8,-12.4,5.8,-4.9;
move -164,-185,8.8,-12.4,5.8,-4.9;
move -165,-183.2,8.7,-12.8,5.9,-4.9;
move -165,-181.4,8.7,-12.8,5.9,-4.8;
move -166,-179.4,8.6,-12.8,6,-4.8;
move -167,-177.3,8.6,-12.8,6,-4.7;
move -167,-175.2,8.5,-12.8,6,-4.7;
move -168,-172.9,8.4,-12.8,6.1,-4.6;
move -168,-170.6,8.4,-12.8,6.1,-4.6;
move -169,-168.1,8.3,-12.8,6.2,-4.5;
move -170,-165.6,8.2,-12.8,6.2,-4.5;
move -171,-163,8.1,-13.2,6.2,-4.5;
move -172,-160.4,8,-13.2,6.3,-4.4;
move -172,-157.7,8,-13.2,6.3,-4.4;
move -173,-155.1,7.9,-13.2,6.3,-4.3;
move -174,-152.4,7.8,-13.2,6.4,-4.3;
move -175,-149.8,7.7,-13.2,6.4,-4.2;
move -176,-147.2,7.6,-13.6,6.5,-4.2;
move -177,-144.7,7.5,-13.6,6.5,-4.1;
move -177,-142.2,7.4,-13.6,6.5,-4.1;
move -178,-139.7,7.3,-13.6,6.6,-4;
move -179,-137.4,7.2,-13.6,6.6,-4;
move -180,-135.2,7.1,-13.6,6.6,-3.9;
move -180,-132.9,7,-13.6,6.7,-3.9;
move -181,-130.8,6.9,-13.6,6.7,-3.8;
move -182,-128.7,6.8,-14,6.8,-3.8;
move -182,-126.7,6.7,-14,6.8,-3.7;
move -183,-124.7,6.6,-14,6.8,-3.7;
move -183,-122.8,6.5,-14,6.9,-3.6;
move -184,-120.8,6.4,-14,6.9,-3.6;
move -184,-118.9,6.3,-14,6.9,-3.5;
move -184,-117,6.2,-14,7,-3.5;
move -185,-115.1,6.1,-14,7,-3.4;
move -185,-113.2,5.9,-14,7,-3.4;
move -185,-111.2,5.8,-14,7.1,-3.3;
move -186,-109.4,5.7,-14,7.1,-3.3;
move -186,-107.4,5.6,-14,7.1,-3.2;
move -187,-105.5,5.4,-14,7.2,-3.2;
move -187,-103.6,5.3,-14.4,7.2,-3.1;
move -188,-101.5,5.2,-14.4,7.3,-3.1;
move -188,-99.5,5.1,-14.4,7.3,-3;
move -189,-97.4,5,-14.4,7.3,-3;
move -189,-95.3,4.9,-14.4,7.4,-2.9;
move -189,-93.1,4.8,-14.4,7.4,-2.8;
move -190,-91,4.7,-14.4,7.4,-2.8;
move -190,-88.8,4.6,-14.4,7.5,-2.7;
move -190,-86.7,4.5,-14.4,7.5,-2.7;
move -190,-84.6,4.4,-14.4,7.5,-2.6;
move -190,-82.5,4.3,-14.4,7.6,-2.6;
move -190,-80.5,4.2,-14.4,7.6,-2.5;
move -190,-78.5,4.1,-14.4,7.6,-2.4;
move -190,-76.5,4,-14.4,7.7,-2.4;
move -190,-74.7,3.9,-14.4,7.7,-2.3;
move -189,-72.8,3.8,-14.4,7.7,-2.3;
move -189,-71,3.7,-14.4,7.8,-2.2;
move -188,-69.3,3.7,-14.4,7.8,-2.2;
move -188,-67.7,3.6,-14.4,7.8,-2.1;
move -187,-66.1,3.6,-14.4,7.9,-2;
move -187,-64.5,3.5,-14,7.9,-2;
move -186,-63,3.4,-14,7.9,-1.9;
move -185,-61.5,3.4,-14,8,-1.9;
move -185,-60.1,3.3,-14,8,-1.8;
move -184,-58.7,3.2,-14,8,-1.7;
move -183,-57.2,3.2,-14,8.1,-1.7;
move -182,-55.8,3.1,-14,8.1,-1.6;
move -181,-54.5,3.1,-14,8.1,-1.6;
move -181,-53.1,3,-13.6,8.1,-1.5;
move -180,-51.7,3,-13.6,8.2,-1.4;
move -178,-50.3,3,-13.6,8.2,-1.4;
move -177,-49,2.9,-13.6,8.2,-1.3;
move -176,-47.5,2.9,-13.6,8.3,-1.3;
move -175,-46.1,2.9,-13.2,8.3,-1.2;
move -174,-44.6,2.8,-13.2,8.3,-1.1;
move -173,-43.1,2.8,-13.2,8.4,-1.1;
move -172,-41.6,2.8,-13.2,8.4,-1;
move -170,-39.9,2.8,-13.2,8.4,-1;
move -169,-38.2,2.7,-12.8,8.4,-0.9;
move -167,-36.3,2.7,-12.8,8.5,-0.8;
move -166,-34.4,2.7,-12.8,8.5,-0.8;
move -164,-32.4,2.7,-12.8,8.5,-0.7;
move -162,-30.2,2.7,-12.4,8.6,-0.6;
move -160,-28,2.7,-12.4,8.6,-0.6;
move -157,-25.7,2.7,-12.4,8.6,-0.5;
move -155,-23.4,2.6,-12,8.6,-0.4;
move -152,-21,2.6,-11.6,8.7,-0.4;
move -149,-18.5,2.6,-11.6,8.7,-0.3;
move -146,-16,2.6,-11.2,8.7,-0.3;
move -143,-13.4,2.6,-11.2,8.7,-0.2;
move -141,-10.8,2.6,-10.8,8.8,-0.1;
move -138,-8.1,2.6,-10.8,8.8,-0.1;
move -135,-5.5,2.6,-10.4,8.8,0;
move -132,-2.8,2.6,-10.4,8.8,0.1;
move -129,0,2.6,-10,8.8,0.1;
move -125,2.7,2.6,-10,8.9,0.2;
move -122,5.3,2.6,-9.6,8.9,0.3;
move -119,8,2.6,-9.6,8.9,0.3;
move -115,10.6,2.6,-9.2,8.9,0.4;
move -112,13.1,2.6,-8.8,9,0.5;
move -108,15.5,2.6,-8.8,9,0.5;
move -105,17.9,2.6,-8.4,9,0.6;
move -101,20.1,2.6,-8,9,0.7;
move -97,22.1,2.6,-8,9,0.7;
move -93,24.1,2.6,-7.6,9.1,0.8;
move -89,25.8,2.6,-7.2,9.1,0.9;
move -85,27.5,2.6,-7.2,9.1,0.9;
move -81,29,2.6,-6.8,9.1,1;
move -77,30.3,2.6,-6.4,9.1,1.1;
move -73,31.4,2.6,-6,9.1,1.1;
move -69,32.4,2.6,-6,9.2,1.2;
move -64,33.2,2.6,-5.6,9.2,1.3;
move -60,33.9,2.6,-5.2,9.2,1.3;
move -56,34.5,2.6,-4.8,9.2,1.4;
move -51,34.9,2.6,-4.8,9.2,1.5;
move -47,35.2,2.6,-4.4,9.2,1.5;
move -42,35.4,2.6,-4,9.2,1.6;
move -38,35.6,2.6,-3.6,9.3,1.7;
move -33,35.6,2.6,-3.2,9.3,1.7;
move -28,35.6,2.6,-3.2,9.3,1.8;
move -24,35.4,2.6,-2.8,9.3,1.9;
move -19,35.3,2.6,-2.4,9.3,1.9;
move -15,35.1,2.6,-2,9.3,2;
move -10,34.8,2.6,-1.6,9.3,2.1;
move -5,34.5,2.7,-1.2,9.3,2.1;
move -1,34.2,2.7,-1.2,9.3,2.2;
move 4,33.9,2.7,-0.8,9.3,2.3;
move 9,33.5,2.7,-0.4,9.3,2.3;
move 13,33.2,2.8,-0,9.4,2.4;
move 18,32.8,2.8,0.4,9.4,2.5;
move 22,32.4,2.8,0.4,9.4,2.6;
move 26,32,2.8,0.8,9.4,2.6;
move 31,31.6,2.9,1.2,9.4,2.7;
move 35,31.3,2.9,1.6,9.4,2.8;
move 40,30.9,2.9,1.6,9.4,2.8;
move 44,30.6,3,2,9.4,2.9;
move 49,30.3,3,2.4,9.4,3;
move 54,30,3.1,2.8,9.4,3;
move 58,29.7,3.1,3.2,9.4,3.1;
move 62,29.3,3.1,3.6,9.4,3.2;
move 67,29,3.2,3.6,9.4,3.2;
move 71,28.6,3.2,4,9.4,3.3;
move 75,28.2,3.3,4.4,9.4,3.4;
move 79,27.8,3.3,4.8,9.4,3.4;
move 83,27.3,3.4,4.8,9.4,3.5;
move 87,26.7,3.4,5.2,9.4,3.6;
move 91,26.2,3.5,5.2,9.4,3.7;
move 94,25.5,3.5,5.6,9.4,3.7;
move 98,24.8,3.6,6,9.4,3.8;
move 101,24.1,3.6,6,9.4,3.9;
move 105,23.3,3.7,6.4,9.3,3.9;
move 108,22.4,3.8,6.8,9.3,4;
move 112,21.5,3.8,6.8,9.3,4.1;
move 115,20.5,3.9,7.2,9.3,4.1;
move 118,19.4,3.9,7.2,9.3,4.2;
move 122,18.3,4,7.6,9.3,4.3;
move 125,17.1,4.1,7.6,9.3,4.3;
move 128,15.8,4.1,8,9.3,4.4;
move 131,14.5,4.2,8.4,9.3,4.5;
move 134,13.2,4.3,8.4,9.2,4.5;
move 137,11.8,4.3,8.8,9.2,4.6;
move 140,10.4,4.4,8.8,9.2,4.7;
move 143,9,4.5,9.2,9.2,4.7;
move 146,7.5,4.5,9.2,9.2,4.8;
move 149,6.1,4.6,9.6,9.2,4.9;
move 152,4.7,4.7,9.6,9.2,4.9;
move 154,3.2,4.7,10,9.1,5;
move 157,1.8,4.8,10,9.1,5.1;
move 159,0.4,4.9,10.4,0,5.2;
move 161,-1,5,10.4,0,5.2;
move 163,-2.4,5,10.4,0,5.3;
move 165,-3.8,5.1,10.8,0,5.4;
move 167,-5.2,5.2,10.8,0,5.4;
move 169,-6.6,5.2,10.8,0,5.5;
move 170,-7.9,5.3,10.8,0,5.6;
move 172,-9.3,5.3,11.2,0,5.6;
move 173,-10.7,5.4,11.2,0,5.7;
move 174,-12,5.5,11.2,0,5.7;
move 176,-13.4,5.5,11.6,0,5.8;
move 177,-14.8,5.6,11.6,0,5.9;
move 177,-16.2,5.6,11.6,0,5.9;
move 178,-17.6,5.7,11.6,0,6;
move 178,-19,5.7,11.6,0,6.1;
move 179,-20.5,5.7,11.6,0,6.1;
move 179,-22.1,5.8,11.6,0,6.2;
move 179,-23.6,5.9,11.6,0,6.3;
move 179,-25.3,5.9,11.6,0,6.3;
move 179,-27.1,6,11.6,0,6.4;
move 179,-29.1,6,11.6,0,6.4;
move 179,-31.1,6,11.6,0,6.5;
move 178,-33.2,6.1,11.6,0,6.6;
move 178,-35.4,6.1,11.6,0,6.6;
move 177,-37.8,6.1,11.6,0,6.7;
move 176,-40.2,6.1,11.6,0,6.8;
move 175,-42.8,6.1,11.2,0,6.8;
move 174,-45.5,6.1,11.2,0,6.9;
move 172,-48.2,6.1,11.2,0,6.9;
move 171,-51,6.1,11.2,0,7;
move 169,-53.9,6.1,10.8,0,7.1;
move 167,-56.9,6.1,10.8,0,7.1;
move 166,-60,6,10.8,0,7.2;
move 164,-63.1,6,10.4,0,7.2;
move 162,-66.2,6,10.4,0,7.3;
move 159,-69.3,5.9,10.4,0,7.4;
move 157,-72.4,5.9,10,7.8,7.4;
move 155,-75.4,5.8,10,7.8,7.5;
move 152,-78.4,5.8,9.6,7.7,7.5;
move 149,-81.3,5.7,9.6,7.7,7.6;
move 146,-84.1,5.6,9.2,7.6,7.6;
move 144,-86.8,5.6,9.2,7.6,7.7;
move 141,-89.3,5.5,8.8,7.5,7.7;
move 138,-91.7,5.4,8.8,7.5,7.8;
move 135,-93.8,5.3,8.4,7.4,7.9;
move 131,-95.8,5.2,8.4,7.3,7.9;
move 128,-97.5,5.2,8,7.3,8;
move 125,-99,5.1,7.6,7.2,8;
move 121,-100.3,5,7.6,7.2,8.1;
move 118,-101.4,4.9,7.2,7.1,8.1;
move 115,-102.2,4.7,7.2,7,8.2;
move 111,-102.9,4.6,6.8,7,8.2;
move 108,-103.4,4.5,6.4,6.9,8.3;
move 105,-103.8,4.4,6.4,6.9,8.3;
move 101,-104,4.3,6,6.8,8.4;
move 98,-104.1,4.2,6,6.7,8.4;
move 94,-104.1,4.1,5.6,6.7,8.5;
move 91,-104.1,3.9,5.2,6.6,8.5;
move 87,-104,3.8,5.2,6.5,8.6;
move 84,-103.9,3.7,4.8,6.4,8.6;
move 80,-103.7,3.6,4.8,6.4,8.7;
move 77,-103.6,3.5,4.4,6.3,8.7;
move 73,-103.6,3.3,4,6.2,8.8;
move 70,-103.5,3.2,4,6.2,8.8;
move 67,-103.5,3.1,3.6,6.1,8.8;
move 63,-103.4,3,3.2,6,8.9;
move 60,-103.4,2.8,3.2,5.9,8.9;
move 57,-103.5,2.7,2.8,5.9,9;
move 53,-103.5,2.6,2.8,5.8,9;
move 50,-103.5,2.5,2.4,5.7,9.1;
move 47,-103.4,2.4,2.4,5.6,9.1;
move 44,-103.4,2.3,2,5.6,9.1;
move 41,-103.3,2.2,2,5.5,9.2;
move 38,-103.3,2.1,1.6,5.4,9.2;
move 35,-103.2,2,1.2,5.3,9.3;
move 33,-103,1.9,1.2,5.2,9.3;
move 30,-102.9,1.8,1.2,5.2,9.3;
move 27,-102.8,1.7,0.8,5.1,9.4;
move 25,-102.6,1.6,0.8,5,9.4;
move 22,-102.5,1.5,0.4,4.9,9.4;
move 20,-102.3,1.4,0.4,4.8,9.5;
move 18,-102,1.3,0,4.7,9.5;
move 15,-101.8,1.2,0,4.6,9.5;
move 13,-101.5,1.2,-0,4.6,9.6;
move 11,-101.2,1.1,-0.4,4.5,9.6;
move 10,-100.9,1,-0.4,4.4,9.6;
move 8,-100.6,1,-0.4,4.3,9.7;
move 6,-100.3,0.9,-0.8,4.2,9.7;
move 5,-99.9,0.8,-0.8,4.1,9.7;
move 3,-99.5,0.8,-0.8,4,9.7;
move 2,-99,0.7,-0.8,3.9,9.8;
move 0,-98.5,0.6,-1.2,3.8,9.8;
move -1,-97.9,0.6,-1.2,3.7,9.8;
move -2,-97.3,0.5,-1.2,3.6,9.8;
move -3,-96.7,0.4,-1.2,3.5,9.8;
move -4,-96,0.4,-1.2,3.5,9.9;
move -5,-95.3,0.3,-1.6,3.4,9.9;
move -6,-94.5,0.3,-1.6,3.3,9.9;
move -7,-93.8,0.2,-1.6,3.2,9.9;
move -7,-92.9,0.2,-1.6,3.1,9.9;
move -8,-92.1,0.2,-1.6,3,9.9;
move -9,-91.2,0.1,-1.6,2.9,9.9;
move -9,-90.3,0.1,-1.6,2.8,9.9;
move -10,-89.4,0,-1.6,2.7,9.9;
move -10,-88.4,-0,-1.6,2.6,9.9;
move -10,-87.5,-0.1,-2,2.5,10;
move -10,-86.6,-0.1,-2,2.4,10;
move -10,-85.6,-0.2,-2,2.3,10;
move -10,-84.7,-0.2,-2,2.2,10;
move -10,-83.8,-0.3,-1.6,2,10;
move -10,-82.9,-0.3,-1.6,1.9,10;
move -10,-82.1,-0.4,-1.6,1.8,10;
move -9,-81.2,-0.4,-1.6,1.7,10;
move -9,-80.5,-0.5,-1.6,1.6,10;
move -9,-79.8,-0.5,-1.6,1.5,10;
move -9,-79.2,-0.6,-1.6,1.4,10;
move -9,-78.7,-0.7,-1.6,1.3,10;
move -9,-78.3,-0.7,-1.6,1.2,10;
move -9,-78,-0.8,-2,1.1,10;
move -9,-77.8,-0.8,-2,1,10;
move -9,-77.7,-0.9,-1.6,0.9,10;
move -9,-77.7,-1,-1.6,0.8,10;
move -8,-77.9,-1,-1.6,0.6,10;
move -8,-78.1,-1.1,-1.6,0.5,10;
move -8,-78.4,-1.2,-1.6,0.4,10;
move -7,-78.8,-1.3,-1.6,0.3,10;
move -6,-79.3,-1.3,-1.6,0.2,10;
move -6,-79.8,-1.4,-1.6,0.1,10;
move -5,-80.5,-1.5,-1.2,-0,10;
move -4,-81.1,-1.6,-1.2,-0.1,10;
move -4,-81.8,-1.6,-1.2,-0.3,10;
move -4,-82.5,-1.7,-1.2,-0.4,10;
move -3,-83.2,-1.8,-1.2,-0.5,10;
move -3,-83.9,-1.9,-1.2,-0.6,10;
move -3,-84.6,-1.9,-1.2,-0.7,10;
move -3,-85.2,-2,-1.2,-0.8,10;
move -3,-85.8,-2.1,-1.2,-0.9,10;
move -2,-86.4,-2.2,-1.2,-1.1,10;
move -2,-87,-2.2,-1.2,-1.2,10;
move -2,-87.4,-2.3,-1.2,-1.3,10;
move -2,-87.9,-2.4,-1.2,-1.4,10;
move -2,-88.3,-2.4,-1.2,-1.5,10;
move -2,-88.6,-2.5,-1.2,-1.7,10;
move -2,-88.8,-2.6,-1.2,-1.8,10;
move -2,-88.9,-2.6,-1.2,-1.9,10;
move -2,-89,-2.7,-1.2,-2,10;
move -2,-89.1,-2.8,-1.2,-2.1,10;
move -2,-89.1,-2.8,-1.2,-2.2,10;
move -2,-89,-2.9,-1.2,-2.4,10;
move -2,-88.9,-3,-1.2,-2.5,10;
move -2,-88.8,-3,-1.2,-2.6,10;
move -2,-88.6,-3.1,-1.2,-2.7,10;
move -3,-88.3,-3.1,-1.2,-2.8,9.9;
move -3,-88,-3.2,-1.2,-3,9.9;
move -3,-87.6,-3.2,-1.2,-3.1,9.9;
move -3,-87.2,-3.2,-1.2,-3.2,9.9;
move -3,-86.7,-3.3,-1.2,-3.3,9.9;
move -3,-86.2,-3.3,-1.2,-3.4,9.9;
move -4,-85.6,-3.4,-1.2,-3.6,9.9;
move -5,-85,-3.4,-1.2,-3.7,9.9;
move -5,-84.3,-3.5,-1.2,-3.8,9.9;
move -6,-83.6,-3.5,-1.6,-3.9,9.8;
move -7,-82.9,-3.5,-1.6,-4,9.8;
move -8,-82.1,-3.5,-1.6,-4.2,9.8;
move -9,-81.3,-3.5,-1.6,-4.3,9.8;
move -10,-80.4,-3.5,-1.6,-4.4,9.8;
move -11,-79.6,-3.6,-1.6,-4.5,9.7;
move -12,-78.8,-3.6,-2,-4.6,9.7;
move -13,-78,-3.6,-2,-4.7,9.7;
move -14,-77.1,-3.6,-2,-4.9,9.7;
move -15,-76.4,-3.6,-2.4,-5,9.6;
move -16,-75.6,-3.6,-2.4,-5.1,9.6;
move -16,-74.9,-3.5,-2.4,-5.2,9.6;
move -17,-74.2,-3.5,-2,-5.3,9.5;
move -18,-73.7,-3.5,-2,-5.5,9.5;
move -19,-73.1,-3.5,-2,-5.6,9.5;
move -20,-72.6,-3.4,-2.4,-5.7,9.4;
move -21,-72.2,-3.4,-2.4,-5.8,9.4;
move -22,-71.8,-3.4,-2.8,-5.9,9.3;
move -23,-71.5,-3.3,-2.8,-6.1,9.3;
move -25,-71.2,-3.3,-2.8,-6.2,9.3;
move -26,-71.1,-3.3,-2.8,-6.3,9.2;
move -28,-71,-3.2,-2.8,-6.4,9.2;
move -29,-70.9,-3.2,-2.8,-6.5,9.1;
move -31,-71,-3.1,-3.2,-6.6,9.1;
move -32,-71,-3,-3.6,-6.8,9;
move -34,-71.2,-3,-3.6,-6.9,9;
move -35,-71.3,-2.9,-3.6,-7,9;
move -37,-71.5,-2.9,-3.6,-7.1,8.9;
move -38,-71.8,-2.8,-3.6,-7.2,8.9;
move -39,-72,-2.8,-4,-7.3,8.8;
move -40,-72.3,-2.7,-4,-7.4,8.7;
move -41,-72.7,-2.6,-4,-7.6,8.7;
move -42,-73.1,-2.5,-4,-7.7,8.6;
move -43,-73.5,-2.5,-4,-7.8,8.6;
move -44,-74,-2.4,-4,-7.9,8.5;
move -45,-74.4,-2.3,-4,-8,8.5;
move -45,-74.8,-2.2,-4.4,-8.1,8.4;
move -46,-75.2,-2.2,-4.4,-8.2,8.4;
move -47,-75.6,-2.1,-4.4,-8.3,8.3;
move -48,-76,-2,-4.4,-8.5,8.2;
move -49,-76.3,-1.9,-4.4,-8.6,8.2;
move -50,-76.7,-1.8,-4.4,-8.7,8.1;
move -51,-77,-1.8,-4.4,-8.8,8.1;
move -52,-77.3,-1.7,-4.8,-8.9,8;
move -53,-77.5,-1.6,-4.8,-9,7.9;
move -54,-77.7,-1.5,-4.8,-9.1,7.9;
move -55,-77.8,-1.4,-4.8,-9.2,7.8;
move -55,-77.9,-1.4,-4.8,-9.3,7.7;
move -56,-77.9,-1.3,-5.2,-9.4,7.7;
move -57,-77.9,-1.2,-5.2,-9.5,7.6;
move -58,-77.7,-1.2,-5.2,-9.6,7.5;
move -58,-77.5,-1.1,-5.2,-9.7,7.5;
move -58,-77.3,-1,-5.2,-9.8,7.4;
move -59,-77,-0.9,-5.2,-9.9,7.3;
move -59,-76.5,-0.9,-5.2,-10,7.3;
move -58,-75.9,-0.8,-5.2,-10.1,7.2;
move -58,-75.1,-0.8,-5.2,-10.2,7.1;
move -57,-74.1,-0.7,-5.2,-10.3,7.1;
move -56,-72.8,-0.7,-5.2,-10.4,7;
move -55,-71.2,-0.6,-5.2,-10.5,6.9;
move -54,-69.3,-0.6,-4.8,-10.6,6.8;
move -53,-67.2,-0.5,-4.8,-10.7,6.8;
move -51,-64.9,-0.5,-4.8,-10.8,6.7;
move -49,-62.4,-0.4,-4.4,-10.9,6.6;
move -47,-59.7,-0.4,-4.4,-11,6.5;
move -45,-56.8,-0.3,-4.4,-11.1,6.5;
move -42,-53.5,-0.3,-4,-11.2,6.4;
move -39,-49.8,-0.3,-4,-11.3,6.3;
move -36,-45.7,-0.3,-3.6,-11.4,6.2;
move -33,-41.3,-0.3,-3.6,-11.5,6.1;
move -29,-36.8,-0.3,-3.2,-11.5,6.1;
move -25,-32.2,-0.3,-2.8,-11.6,6;
move -21,-27.3,-0.3,-2.8,-11.7,5.9;
move -17,-22.1,-0.3,-2.4,-11.8,5.8;
move -12,-16.7,-0.3,-2,-11.9,5.7;
move -7,-11.2,-0.3,-1.6,-12,5.6;
move -1,-5.5,-0.3,-1.2,-12.1,5.5;
move 5,0.1,-0.3,-0.8,-12.1,5.5;
move 10,5.7,-0.4,-0.4,-12.2,5.4;
move 16,11.1,-0.4,0,-12.3,5.3;
move 23,16.2,-0.4,0.4,-12.4,5.2;
move 29,20.9,-0.4,1.2,-12.5,5.1;
move 35,25.3,-0.5,1.6,-12.5,5;
move 42,29.1,-0.5,2,-12.6,4.9;
move 48,32.5,-0.5,2.4,-12.7,4.8;
move 55,35.3,-0.6,2.8,-12.8,4.8;
move 61,37.6,-0.6,3.2,-12.8,4.7;
move 68,39.2,-0.7,3.6,-12.9,4.6;
move 74,40.3,-0.7,4,-13,4.5;
move 81,40.7,-0.8,4.8,-13,4.4;
move 88,40.4,-0.8,5.2,-13.1,4.3;
move 95,39.4,-0.9,5.6,-13.2,4.2;
move 102,37.6,-0.9,6,-13.2,4.1;
move 110,35,-0.9,6.8,-13.3,4;
move 117,31.7,-1,7.2,-13.4,3.9;
move 124,27.5,-1,7.6,-13.4,3.8;
move 132,22.6,-1,8.4,-13.5,3.7;
move 139,16.9,-1.1,8.8,-13.6,3.6;
move 147,10.3,-1.1,9.2,-13.6,3.5;
move 154,3,-1.1,10,-13.7,3.4;
move 161,-5.1,-1.1,10.4,0,3.3;
move 168,-13.9,-1.1,10.8,0,3.2;
move 175,-23.4,-1.1,11.6,0,3.1;
move 182,-33.4,-1.2,12,0,3;
move 188,-44,-1.2,12.4,0,2.9;
move 194,-55.1,-1.2,12.8,0,2.8;
move 200,-66.5,-1.1,13.2,0,2.7;
move 206,-78.1,-1.1,13.6,0,2.6;
move 211,-89.8,-1.1,14,0,2.5;
move 217,-101.5,-1.1,14.4,0,2.4;
move 222,-113.1,-1,14.8,0,2.3;
move 227,-124.3,-1,14.8,0,2.2;
move 232,-135,-0.9,15.2,0,2.1;
move 236,-145.3,-0.8,15.6,0,2;
move 241,-155,-0.7,16,0,1.9;
move 245,-164.1,-0.6,16.4,0,1.8;
move 249,-172.6,-0.5,16.8,0,1.7;
move 253,-180.5,-0.4,17.2,0,1.6;
move 257,-187.7,-0.3,17.2,0,1.5;
move 260,-194.2,-0.2,17.6,0,1.4;
move 263,-199.8,-0.1,17.6,0,1.3;
move 265,-204.8,0,17.6,0,1.2;
move 268,-209.2,0.2,18,0,1.1;
move 270,-213,0.3,18,0,1;
move 272,-216.4,0.5,18,0,0.9;
move 274,-219.3,0.7,18.4,0,0.8;
move 276,-221.8,0.9,18.4,0,0.7;
move 278,-223.9,1,18.8,0,0.6;
move 280,-225.6,1.2,18.8,0,0.5;
move 281,-227,1.4,18.8,0,0.4;
move 283,-228.2,1.5,18.8,0,0.3;
move 284,-229.2,1.7,19.2,0,0.2;
move 285,-230.1,1.9,19.2,0,0.1;
move 286,-231,2.1,19.2,0,-0.1;
move 286,-231.9,2.3,19.2,0,-0.2;
move 287,-232.9,2.5,19.2,0,-0.3;
move 287,-234,2.7,19.2,0,-0.4;
move 287,-235.2,2.9,19.2,0,-0.5;
move 288,-236.5,3.1,19.2,0,-0.6;
move 288,-238,3.3,19.2,0,-0.7;
move 288,-239.6,3.5,19.2,0,-0.8;
move 287,-241.4,3.7,19.6,0,-0.9;
move 287,-243.3,4,19.2,0,-1;
move 287,-245.3,4.2,19.2,0,-1.1;
move 286,-247.5,4.4,19.2,0,-1.2;
move 285,-249.8,4.6,19.2,0,-1.3;
move 284,-252.3,4.8,19.2,0,-1.4;
move 283,-254.8,4.9,18.8,0,-1.5;
move 282,-257.4,5.1,18.8,0,-1.6;
move 281,-260.1,5.3,18.8,0,-1.7;
move 279,-262.8,5.5,18.8,0,-1.8;
move 278,-265.6,5.7,18.4,0,-1.9;
move 277,-268.4,5.8,18.4,0,-2;
move 275,-271.3,6,18.4,0,-2.1;
move 274,-274.2,6.1,18.4,0,-2.3;
move 272,-277.1,6.3,18,0,-2.4;
move 270,-280.1,6.4,18,0,-2.5;
move 268,-283.1,6.6,18,0,-2.6;
move 266,-286.2,6.7,18,0,-2.7;
move 264,-289.4,6.9,17.6,0,-2.8;
move 261,-292.6,7,17.6,0,-2.9;
move 259,-295.9,7.1,17.2,0,-3;
move 256,-299.3,7.2,16.8,0,-3.1;
move 253,-302.7,7.3,16.8,0,-3.2;
move 251,-306.3,7.4,16.4,0,-3.3;
move 248,-309.9,7.5,16.4,0,-3.4;
move 245,-313.6,7.6,16.4,0,-3.5;
move 243,-317.4,7.7,16,0,-3.6;
move 240,-321.3,7.7,16,0,-3.7;
move 238,-325.2,7.8,15.6,0,-3.8;
move 236,-329,7.9,15.2,0,-3.9;
move 233,-332.8,7.9,15.2,0,-4;
move 231,-336.5,8,15.2,0,-4.1;
move 229,-340.1,8,15.2,0,-4.2;
move 227,-343.4,8,15.2,0,-4.3;
move 225,-346.6,8,14.8,0,-4.4;
move 222,-349.5,8,14.8,0,-4.5;
move 220,-352.1,8,14.4,0,-4.6;
move 217,-354.6,8,14.4,0,-4.7;
move 215,-356.7,8,14,0,-4.8;
move 212,-358.5,8,14,0,-4.9;
move 209,-360,8,13.6,0,-5;
move 206,-361.2,7.9,13.6,0,-5.1;
move 204,-362.2,7.9,13.2,0,-5.2;
move 201,-362.8,7.8,13.2,0,-5.3;
move 198,-363.2,7.8,12.8,0,-5.4;
move 195,-363.4,7.7,12.8,0,-5.5;
move 193,-363.3,7.6,12.4,0,-5.6;
move 190,-362.9,7.6,12.4,0,-5.7;
move 188,-362.3,7.5,12,0,-5.8;
move 185,-361.7,7.4,12,0,-5.9;
move 183,-360.9,7.4,11.6,0,-6;
move 181,-360.2,7.3,11.6,0,-6.1;
move 179,-359.4,7.2,11.6,0,-6.2;
move 176,-358.7,7.1,11.6,0,-6.3;
move 174,-358,7,11.2,0,-6.4;
move 172,-357.5,6.9,11.2,0,-6.5;
move 170,-357,6.9,10.8,0,-6.6;
move 168,-356.7,6.8,10.8,0,-6.6;
move 166,-356.5,6.7,10.8,0,-6.7;
move 164,-356.5,6.6,10.4,0,-6.8;
move 163,-356.8,6.5,10.4,0,-6.9;
move 161,-357.2,6.4,10,-12.6,-7;
move 160,-357.9,6.2,10,-12.5,-7.1;
move 159,-358.8,6.1,10,-12.4,-7.2;
move 158,-359.9,6,10,-12.3,-7.3;
move 158,-361.2,5.9,10,-12.3,-7.4;
move 157,-362.6,5.8,10,-12.2,-7.4;
move 157,-364.1,5.7,10,-12.1,-7.5;
move 157,-365.6,5.5,10,-12,-7.6;
move 157,-367.2,5.4,10,-11.9,-7.7;
move 157,-368.8,5.3,10,-11.8,-7.8;
move 157,-370.3,5.2,10,-11.7,-7.9;
move 157,-371.7,5,10,-11.6,-7.9;
move 157,-373,4.9,10,-11.5,-8;
move 157,-374,4.8,10,-11.4,-8.1;
move 158,-374.8,4.7,10,-11.4,-8.2;
move 158,-375.5,4.5,10,-11.3,-8.3;
move 159,-375.9,4.4,10,-11.2,-8.3;
move 160,-376,4.3,10,-11.1,-8.4;
move 160,-376,4.2,10.4,0,-8.5;
move 161,-375.8,4,10.4,0,-8.6;
move 161,-375.5,3.9,10.8,0,-8.6;
move 161,-375.1,3.8,10.4,0,-8.7;
move 161,-374.7,3.7,10.4,0,-8.8;
move 161,-374.4,3.6,10.4,0,-8.9;
move 160,-374.1,3.5,10.4,0,-8.9;
move 160,-373.9,3.4,10.4,0,-9;
move 159,-373.8,3.3,10,-10.1,-9.1;
move 158,-373.9,3.2,10,-10,-9.1;
move 158,-374.3,3.1,10,-9.9,-9.2;
move 157,-375.1,3,10,-9.8,-9.3;
move 156,-376.2,3,10,-9.7,-9.3;
move 155,-377.8,2.9,10,-9.6,-9.4;
move 154,-379.8,2.8,10,-9.4,-9.5;
move 153,-382.3,2.7,9.6,-9.3,-9.5;
move 152,-385.2,2.7,9.6,-9.2,-9.6;
move 150,-388.6,2.6,9.6,-9.1,-9.7;
move 149,-392.5,2.5,9.6,-9,-9.7;
move 147,-396.8,2.4,9.6,-8.9,-9.8;
move 145,-401.5,2.4,9.2,-8.7,-9.9;
move 143,-406.6,2.3,9.2,-8.6,-9.9;
move 141,-412.1,2.3,8.8,-8.5,-10;
move 139,-418,2.2,8.8,-8.4,-10;
move 137,-424.1,2.2,8.8,-8.3,-10.1;
move 134,-430.4,2.1,8.4,-8.1,-10.2;
move 132,-436.9,2,8.4,-8,-10.2;
move 130,-443.3,2,8,-7.9,-10.3;
move 127,-449.8,1.9,8,-7.8,-10.3;
move 124,-456,1.9,7.6,-7.6,-10.4;
move 122,-462,1.9,7.6,-7.5,-10.4;
move 119,-467.6,1.8,7.2,-7.4,-10.5;
move 117,-472.7,1.8,7.2,-7.3,-10.5;
move 114,-477.3,1.8,7.2,-7.1,-10.6;
move 111,-481.3,1.7,6.8,-7,-10.6;
move 108,-484.5,1.7,6.8,-6.9,-10.7;
move 105,-487.1,1.7,6.4,-6.7,-10.7;
move 102,-488.9,1.7,6,-6.6,-10.8;
move 99,-489.9,1.7,6,-6.5,-10.8;
move 95,-490,1.6,5.6,-6.3,-10.9;
move 92,-489.5,1.6,5.6,-6.2,-10.9;
move 89,-488.1,1.6,5.2,-6.1,-10.9;
move 85,-486.1,1.6,5.2,-5.9,-11;
move 81,-483.4,1.6,4.8,-5.8,-11;
move 77,-480.1,1.6,4.4,-5.7,-11.1;
move 73,-476.2,1.6,4,-5.5,-11.1;
move 70,-472,1.5,4,-5.4,-11.2;
move 66,-467.4,1.6,3.6,-5.3,-11.2;
move 62,-462.7,1.6,3.2,-5.1,-11.2;
move 58,-458,1.6,2.8,-5,-11.3;
move 53,-453.4,1.6,2.8,-4.8,-11.3;
move 49,-449.1,1.6,2.4,-4.7,-11.3;
move 45,-445.2,1.6,2.4,-4.6,-11.4;
move 41,-441.9,1.6,2,-4.4,-11.4;
move 37,-439.2,1.6,1.6,-4.3,-11.5;
move 32,-437.2,1.7,1.2,-4.1,-11.5;
move 28,-435.8,1.7,0.8,-4,-11.5;
move 23,-435.2,1.7,0.8,-3.9,-11.5;
move 19,-435.5,1.7,0.4,-3.7,-11.6;
move 14,-436.7,1.8,-0,-3.6,-11.6;
move 9,-438.7,1.8,-0.4,-3.4,-11.6;
move 4,-441.5,1.8,-0.8,-3.3,-11.7;
move 0,-445.2,1.9,-1.2,-3.2,-11.7;
move -5,-449.5,1.9,-1.6,-3,-11.7;
move -10,-454.5,1.9,-1.6,-2.9,-11.7;
move -14,-459.9,2,-2,-2.7,-11.8;
move -18,-465.6,2,-2.4,-2.6,-11.8;
move -23,-471.5,2,-2.8,-2.4,-11.8;
move -27,-477.5,2.1,-2.8,-2.3,-11.8;
move -31,-483.3,2.1,-3.2,-2.2,-11.8;
move -36,-488.8,2.1,-3.6,-2,-11.9;
move -39,-493.7,2.1,-4,-1.9,-11.9;
move -43,-498.1,2.1,-4.4,-1.7,-11.9;
move -47,-501.6,2.2,-4.4,-1.6,-11.9;
move -50,-504.3,2.2,-4.8,-1.4,-11.9;
move -53,-506.1,2.2,-4.8,-1.3,-11.9;
move -56,-506.8,2.2,-5.2,-1.1,-11.9;
move -59,-506.5,2.3,-5.2,-1,-11.9;
move -61,-505.1,2.3,-5.2,-0.9,-11.9;
move -64,-502.6,2.3,-5.6,-0.7,-11.9;
move -66,-499.2,2.3,-5.6,-0.6,-11.9;
move -68,-494.8,2.3,-6,-0.4,-11.9;
move -70,-489.6,2.3,-6,-0.3,-11.9;
move -73,-483.6,2.3,-6,-0.1,-11.9;
move -75,-476.9,2.3,-6.4,0,-11.9;
move -77,-469.8,2.2,-6.4,0.1,-11.9;
move -79,-462.2,2.2,-6.8,0.3,-11.9;
move -81,-454.4,2.2,-6.8,0.4,-11.9;
move -82,-446.4,2.2,-6.8,0.6,-11.9;
move -84,-438.4,2.1,-7.2,0.7,-11.9;
move -85,-430.5,2.1,-7.2,0.9,-11.9;
move -85,-422.7,2.1,-7.2,1,-11.9;
move -86,-415.3,2.1,-7.2,1.1,-11.9;
move -86,-408.2,2,-7.2,1.3,-11.9;
move -86,-401.5,2,-7.2,1.4,-11.9;
move -86,-395.3,1.9,-7.2,1.6,-11.9;
move -86,-389.5,1.9,-7.2,1.7,-11.8;
move -86,-384.1,1.8,-7.2,1.9,-11.8;
move -85,-379.3,1.7,-7.2,2,-11.8;
move -84,-375,1.7,-6.8,2.1,-11.8;
move -83,-371,1.6,-6.8,2.3,-11.8;
move -82,-367.5,1.5,-6.8,2.4,-11.7;
move -81,-364.3,1.5,-6.8,2.6,-11.7;
move -79,-361.6,1.4,-6.8,2.7,-11.7;
move -77,-359.3,1.3,-6.8,2.8,-11.7;
move -76,-357.5,1.2,-6.4,3,-11.6;
move -73,-356,1.1,-6.4,3.1,-11.6;
move -71,-354.8,1,-6,3.3,-11.6;
move -68,-353.9,1,-6,3.4,-11.6;
move -66,-353.3,0.9,-5.6,3.5,-11.5;
move -63,-352.8,0.8,-5.6,3.7,-11.5;
move -59,-352.4,0.7,-5.2,3.8,-11.5;
move -56,-352.2,0.6,-5.2,3.9,-11.4;
move -52,-352.1,0.5,-4.8,4.1,-11.4;
move -49,-352.1,0.4,-4.4,4.2,-11.4;
move -45,-352.3,0.3,-4.4,4.3,-11.3;
move -40,-352.5,0.1,-4,4.5,-11.3;
move -36,-352.9,0,-3.6,4.6,-11.2;
move -32,-353.2,-0.1,-3.2,4.7,-11.2;
move -28,-353.7,-0.2,-2.8,4.9,-11.2;
move -23,-354.2,-0.4,-2.8,5,-11.1;
move -18,-354.8,-0.5,-2.4,5.1,-11.1;
move -14,-355.4,-0.6,-2,5.3,-11;
move -9,-356,-0.8,-1.6,5.4,-11;
move -5,-356.7,-0.9,-1.2,5.5,-11;
move 0,-357.5,-1,-1.2,5.6,-10.9;
move 4,-358.2,-1.2,-0.8,5.8,-10.9;
move 9,-358.9,-1.3,-0.4,5.9,-10.8;
move 14,-359.7,-1.4,-0,6,-10.8;
move 18,-360.4,-1.6,0.4,6.1,-10.7;
move 22,-361.1,-1.7,0.8,6.3,-10.7;
move 26,-361.8,-1.8,0.8,6.4,-10.6;
move 30,-362.5,-1.9,1.2,6.5,-10.6;
move 34,-363.2,-2,1.6,6.6,-10.5;
move 38,-363.8,-2.1,1.6,6.8,-10.5;
move 42,-364.5,-2.2,2,6.9,-10.4;
move 45,-365.1,-2.3,2.4,7,-10.4;
move 48,-365.6,-2.4,2.4,7.1,-10.3;
move 51,-366.1,-2.5,2.8,7.2,-10.3;
move 55,-366.6,-2.5,2.8,7.3,-10.2;
move 58,-367.1,-2.6,2.8,7.5,-10.2;
move 61,-367.5,-2.7,3.2,7.6,-10.1;
move 64,-367.9,-2.8,3.6,7.7,-10.1;
move 67,-368.3,-2.8,3.6,7.8,-10;
move 69,-368.6,-2.9,4,7.9,-9.9;
move 72,-369,-2.9,4,8,-9.9;
move 75,-369.3,-3,4.4,8.1,-9.8;
move 78,-369.7,-3.1,4.4,8.3,-9.8;
move 81,-370.2,-3.1,4.8,8.4,-9.7;
move 84,-370.7,-3.2,4.8,8.5,-9.6;
move 87,-371.2,-3.2,5.2,8.6,-9.6;
move 90,-371.7,-3.2,5.2,8.7,-9.5;
move 94,-372.4,-3.3,5.6,8.8,-9.4;
move 97,-373,-3.3,5.6,8.9,-9.4;
move 100,-373.7,-3.4,6,9,-9.3;
move 103,-374.5,-3.4,6.4,9.1,-9.2;
move 106,-375.4,-3.4,6.4,9.2,-9.2;
move 109,-376.4,-3.4,6.8,9.3,-9.1;
move 112,-377.5,-3.5,7.2,9.4,-9;
move 115,-378.7,-3.5,7.2,9.5,-9;
move 117,-380,-3.5,7.2,9.6,-8.9;
move 119,-381.5,-3.4,7.6,9.7,-8.8;
move 121,-383.1,-3.4,7.6,9.8,-8.8;
move 123,-384.8,-3.4,7.6,9.9,-8.7;
move 124,-386.7,-3.4,8,10,-8.6;
move 126,-388.8,-3.4,8,10.1,-8.5;
move 127,-390.9,-3.4,8,10.1,-8.5;
move 128,-393.2,-3.4,8,10.2,-8.4;
move 129,-395.6,-3.3,8,10.3,-8.3;
move 130,-398,-3.3,8,10.4,-8.2;
move 130,-400.6,-3.3,8,10.5,-8.2;
move 131,-403.2,-3.3,8.4,10.6,-8.1;
move 132,-405.8,-3.2,8.4,10.7,-8;
move 132,-408.5,-3.2,8.4,10.7,-7.9;
move 133,-411.1,-3.1,8.4,10.8,-7.9;
move 133,-413.6,-3.1,8.4,10.9,-7.8;
move 133,-416.1,-3,8.4,11,-7.7;
move 134,-418.4,-3,8.4,11.1,-7.6;
move 134,-420.7,-2.9,8.4,11.1,-7.5;
move 134,-422.8,-2.9,8.4,11.2,-7.5;
move 134,-424.8,-2.8,8.4,11.3,-7.4;
move 134,-426.6,-2.8,8.4,11.4,-7.3;
move 134,-428.2,-2.7,8.4,11.4,-7.2;
move 133,-429.7,-2.6,8.4,11.5,-7.1;
move 133,-431,-2.6,8.4,11.6,-7;
move 133,-432.2,-2.5,8.4,11.6,-7;
move 132,-433.2,-2.5,8.4,11.7,-6.9;
move 132,-434.1,-2.4,8.4,11.8,-6.8;
move 131,-434.9,-2.3,8.4,11.8,-6.7;
move 131,-435.5,-2.3,8,11.9,-6.6;
move 130,-436,-2.2,8,12,-6.5;
move 130,-436.4,-2.1,8,12,-6.4;
move 129,-436.7,-2.1,8,12.1,-6.3;
move 129,-437,-2,8,12.1,-6.3;
move 128,-437.2,-2,8,12.2,-6.2;
move 127,-437.3,-1.9,8,12.3,-6.1;
move 127,-437.4,-1.8,8,12.3,-6;
move 126,-437.5,-1.7,8,12.4,-5.9;
move 125,-437.5,-1.7,8,12.4,-5.8;
move 124,-437.6,-1.6,7.6,12.5,-5.7;
move 123,-437.8,-1.5,7.6,12.5,-5.6;
move 122,-438,-1.5,7.6,12.6,-5.5;
move 121,-438.4,-1.4,7.6,12.6,-5.4;
move 120,-438.8,-1.4,7.2,12.7,-5.3;
move 119,-439.3,-1.3,7.2,12.7,-5.3;
move 119,-440,-1.3,7.2,12.7,-5.2;
move 118,-440.8,-1.2,7.2,12.8,-5.1;
move 117,-441.7,-1.2,7.2,12.8,-5;
move 117,-442.7,-1.1,7.2,12.9,-4.9;
move 116,-443.9,-1,7.2,12.9,-4.8;
move 116,-445.1,-1,7.2,12.9,-4.7;
move 115,-446.5,-0.9,7.2,13,-4.6;
move 115,-448,-0.9,7.2,13,-4.5;
move 114,-449.6,-0.8,7.2,13,-4.4;
move 114,-451.2,-0.7,6.8,13.1,-4.3;
move 113,-452.9,-0.7,6.8,13.1,-4.2;
move 112,-454.6,-0.6,6.8,13.1,-4.1;
move 111,-456.3,-0.6,6.8,13.2,-4;
move 110,-458,-0.5,6.8,13.2,-3.9;
move 110,-459.7,-0.4,6.8,13.2,-3.8;
move 109,-461.3,-0.4,6.8,13.2,-3.7;
move 108,-462.9,-0.3,6.4,13.3,-3.6;
move 108,-464.3,-0.3,6.4,13.3,-3.5;
move 107,-465.6,-0.2,6.4,13.3,-3.5;
move 106,-466.8,-0.2,6.4,13.3,-3.4;
move 106,-467.9,-0.1,6.4,13.3,-3.3;
move 105,-468.8,-0,6.4,13.4,-3.2;
move 105,-469.5,0,6.4,13.4,-3.1;
move 104,-470.1,0.1,6.4,13.4,-3;
move 104,-470.5,0.1,6.4,13.4,-2.9;
move 103,-470.8,0.2,6.4,13.4,-2.8;
move 102,-470.9,0.2,6,13.4,-2.7;
move 102,-470.8,0.3,6,13.4,-2.6;
move 101,-470.7,0.3,6,13.4,-2.5;
move 101,-470.4,0.4,6,13.4,-2.4;
move 101,-470.1,0.4,6,13.4,-2.3;
move 100,-469.7,0.5,6,13.4,-2.2;
move 100,-469.3,0.5,6,13.4,-2.1;
move 100,-468.8,0.6,6,13.4,-2;
move 100,-468.4,0.6,6,13.4,-1.9;
move 99,-468,0.7,6,13.4,-1.8;
move 99,-467.7,0.7,6,13.4,-1.7;
move 99,-467.5,0.8,6,13.4,-1.6;
move 98,-467.3,0.8,6,13.4,-1.5;
move 98,-467.3,0.9,6,13.4,-1.4;
move 97,-467.3,0.9,6,13.4,-1.3;
move 97,-467.6,1,5.6,13.4,-1.2;
move 96,-467.9,1,5.6,13.4,-1.1;
move 96,-468.5,1.1,5.6,13.4,-1;
move 95,-469.1,1.1,5.6,13.4,-0.9;
move 95,-469.8,1.1,5.6,13.4,-0.8;
move 94,-470.7,1.2,5.6,13.3,-0.7;
move 94,-471.7,1.2,5.6,13.3,-0.7;
move 94,-472.8,1.3,5.6,13.3,-0.6;
move 94,-474,1.3,5.6,13.3,-0.5;
move 93,-475.3,1.3,5.6,13.3,-0.4;
move 93,-476.6,1.3,5.6,13.2,-0.3;
move 92,-478.1,1.4,5.6,13.2,-0.2;
move 91,-479.6,1.4,5.6,13.2,-0.1;
move 91,-481.1,1.4,5.2,13.2,0;
move 90,-482.6,1.4,5.2,13.2,0.1;
move 89,-484.1,1.5,5.2,13.1,0.2;
move 88,-485.6,1.5,5.2,13.1,0.3;
move 87,-487.1,1.5,5.2,13.1,0.4;
move 86,-488.7,1.5,5.2,13,0.5;
move 85,-490.1,1.6,4.8,13,0.6;
move 83,-491.6,1.6,4.8,13,0.7;
move 82,-492.9,1.6,4.8,12.9,0.8;
move 81,-494.1,1.6,4.8,12.9,0.9;
move 80,-495.3,1.6,4.4,12.9,1;
move 78,-496.5,1.6,4.4,12.8,1.1;
move 77,-497.5,1.6,4.4,12.8,1.2;
move 76,-498.5,1.6,4.4,12.8,1.2;
move 75,-499.4,1.6,4.4,12.7,1.3;
move 74,-500.3,1.6,4,12.7,1.4;
move 72,-501.1,1.6,4,12.6,1.5;
move 71,-501.8,1.6,4,12.6,1.6;
move 70,-502.4,1.5,4,12.5,1.7;
move 68,-503,1.5,4,12.5,1.8;
move 67,-503.5,1.5,3.6,12.5,1.9;
move 66,-504,1.5,3.6,12.4,2;
move 64,-504.5,1.4,3.6,12.4,2.1;
move 62,-504.8,1.4,3.2,12.3,2.2;
move 61,-505.2,1.4,3.2,12.3,2.2;
move 59,-505.5,1.3,3.2,12.2,2.3;
move 58,-505.8,1.3,3.2,12.2,2.4;
move 56,-506,1.2,2.8,12.1,2.5;
move 54,-506.1,1.2,2.8,12,2.6;
move 52,-506.3,1.2,2.8,12,2.7;
move 51,-506.4,1.1,2.4,11.9,2.8;
move 49,-506.4,1.1,2.4,11.9,2.9;
move 47,-506.5,1.1,2.4,11.8,3;
move 45,-506.5,1,2,11.8,3;
move 43,-506.5,1,2,11.7,3.1;
move 41,-506.4,0.9,2,11.6,3.2;
move 40,-506.4,0.9,1.6,11.6,3.3;
move 38,-506.3,0.8,1.6,11.5,3.4;
move 36,-506.1,0.8,1.6,11.5,3.5;
move 35,-506,0.7,1.2,11.4,3.6;
move 33,-505.9,0.7,1.2,11.3,3.6;
move 32,-505.8,0.6,1.2,11.3,3.7;
move 30,-505.7,0.6,1.2,11.2,3.8;
move 29,-505.6,0.5,0.8,11.1,3.9;
move 28,-505.4,0.4,0.8,11.1,4;
move 27,-505.3,0.4,0.8,11,4.1;
move 26,-505.2,0.3,0.8,10.9,4.1;
move 25,-505.1,0.3,0.8,10.9,4.2;
move 24,-505,0.2,0.8,10.8,4.3;
move 23,-504.9,0.2,0.4,10.7,4.4;
move 22,-504.8,0.1,0.4,10.6,4.4;
move 22,-504.8,0,0.4,10.6,4.5;
move 21,-504.7,-0,0.4,10.5,4.6;
move 20,-504.6,-0.1,0.4,10.4,4.7;
move 20,-504.4,-0.2,0.4,10.3,4.8;
move 19,-504.3,-0.2,0.4,10.3,4.8;
move 18,-504.1,-0.3,0.4,10.2,4.9;
move 18,-504,-0.3,0.4,10.1,5;
move 17,-503.9,-0.4,0,10,5;
move 17,-503.7,-0.4,0,10,5.1;
move 16,-503.5,-0.4,0,9.9,5.2;
move 16,-503.2,-0.5,0,9.8,5.3;
move 15,-503,-0.5,0,9.7,5.3;
move 15,-502.6,-0.6,0,9.6,5.4;
move 15,-502.3,-0.6,0,9.6,5.5;
move 15,-501.8,-0.7,0,9.5,5.5;
move 16,-501.4,-0.7,0,9.4,5.6;
move 16,-500.8,-0.8,0,9.3,5.7;
move 17,-500.3,-0.8,0,9.2,5.8;
move 17,-499.7,-0.8,0,9.1,5.8;
move 18,-499,-0.9,0.4,9.1,5.9;
move 18,-498.4,-0.9,0.4,9,6;
move 19,-497.6,-0.9,0.4,8.9,6;
move 20,-496.8,-1,0.4,8.8,6.1;
move 20,-496,-1,0.4,8.7,6.1;
move 21,-495.2,-1,0.4,8.6,6.2;
move 22,-494.4,-1,0.4,8.5,6.3;
move 23,-493.5,-1.1,0.4,8.4,6.3;
move 23,-492.7,-1.1,0.4,8.4,6.4;
move 24,-492,-1.1,0.8,8.3,6.5;
move 25,-491.2,-1.1,0.8,8.2,6.5;
move 27,-490.6,-1.1,0.8,8.1,6.6;
move 28,-490,-1.1,0.8,8,6.6;
move 29,-489.5,-1.1,1.2,7.9,6.7;
move 30,-489,-1.2,1.2,7.8,6.7;
move 31,-488.8,-1.2,1.2,7.7,6.8;
move 32,-488.6,-1.2,1.2,7.6,6.9;
move 33,-488.6,-1.2,1.2,7.5,6.9;
move 34,-488.7,-1.2,1.2,7.5,7;
move 36,-488.9,-1.2,1.6,7.4,7;
move 37,-489.3,-1.2,1.6,7.3,7.1;
move 38,-489.8,-1.2,1.6,7.2,7.1;
move 39,-490.4,-1.2,1.6,7.1,7.2;
move 40,-491.2,-1.1,2,7,7.2;
move 42,-492.2,-1.1,2,6.9,7.3;
move 43,-493.1,-1.1,2,6.8,7.3;
move 44,-494.2,-1.1,2,6.7,7.4;
move 45,-495.4,-1.1,2,6.6,7.4;
move 46,-496.6,-1,2.4,6.5,7.5;
move 47,-497.8,-1,2.4,6.4,7.5;
move 47,-499,-1,2.4,6.3,7.6;
move 48,-500.3,-1,2.4,6.2,7.6;
move 49,-501.6,-1,2.4,6.1,7.7;
move 49,-502.9,-0.9,2.4,6,7.7;
move 50,-504.2,-0.9,2.4,5.9,7.8;
move 51,-505.5,-0.9,2.4,5.8,7.8;
move 51,-506.7,-0.8,2.4,5.8,7.9;
move 52,-507.9,-0.8,2.8,5.7,7.9;
move 52,-509,-0.8,2.8,5.6,8;
move 53,-510.1,-0.8,2.8,5.5,8;
move 53,-511.1,-0.7,2.8,5.4,8;
move 54,-512.1,-0.7,2.8,5.3,8.1;
move 54,-513,-0.7,2.8,5.2,8.1;
move 54,-513.8,-0.6,2.8,5.1,8.2;
move 54,-514.6,-0.6,2.8,5,8.2;
move 54,-515.3,-0.6,2.8,4.9,8.2;
move 53,-516,-0.5,2.8,4.8,8.3;
move 53,-516.6,-0.5,2.8,4.7,8.3;
move 52,-517.2,-0.5,2.8,4.6,8.4;
move 52,-517.7,-0.5,2.8,4.5,8.4;
move 51,-518.1,-0.4,2.4,4.4,8.4;
move 50,-518.5,-0.4,2.4,4.3,8.5;
move 50,-518.9,-0.4,2.4,4.2,8.5;
move 49,-519.2,-0.3,2.4,4.1,8.5;
move 48,-519.4,-0.3,2.4,4,8.5;
move 48,-519.7,-0.3,2.4,3.9,8.6;
move 47,-519.9,-0.2,2.4,3.8,8.6;
move 46,-520.1,-0.2,2.4,3.7,8.6;
move 45,-520.2,-0.2,2,3.6,8.7;
move 44,-520.3,-0.2,2,3.5,8.7;
move 43,-520.5,-0.1,2,3.4,8.7;
move 42,-520.6,-0.1,2,3.3,8.7;
move 41,-520.8,-0.1,2,3.2,8.8;
move 40,-520.9,-0,2,3.1,8.8;
move 39,-521.1,-0,1.6,3,8.8;
move 38,-521.2,0,1.6,3,8.8;
move 37,-521.4,0,1.6,2.9,8.8;
move 36,-521.5,0.1,1.6,2.8,8.9;
move 35,-521.7,0.1,1.6,2.7,8.9;
move 34,-521.9,0.1,1.2,2.6,8.9;
move 33,-522.1,0.2,1.2,2.5,8.9;
move 32,-522.3,0.2,1.2,2.4,8.9;
move 30,-522.5,0.2,1.2,2.3,8.9;
move 29,-522.7,0.2,1.2,2.2,8.9;
move 28,-522.9,0.2,0.8,2.1,8.9;
move 27,-523.1,0.3,0.8,2,8.9;
move 25,-523.3,0.3,0.8,1.9,8.9;
move 24,-523.5,0.3,0.8,1.8,9;
move 23,-523.6,0.3,0.4,1.7,9;
move 22,-523.8,0.4,0.4,1.6,9;
move 20,-523.9,0.4,0.4,1.5,9;
move 19,-524.1,0.4,0.4,1.5,9;
move 18,-524.2,0.4,0.4,1.4,9;
move 17,-524.3,0.4,0,1.3,9;
move 15,-524.3,0.4,0,1.2,9;
move 14,-524.3,0.4,-0,1.1,9;
move 13,-524.3,0.5,-0,1,9;
move 12,-524.3,0.5,-0.4,0.9,9;
move 11,-524.3,0.5,-0.4,0.8,9;
move 10,-524.2,0.5,-0.4,0.7,9;
move 8,-524.1,0.5,-0.4,0.6,9;
move 7,-524,0.5,-0.4,0.5,9;
move 6,-523.8,0.5,-0.4,0.5,9;
move 5,-523.6,0.5,-0.8,0.4,9;
move 4,-523.3,0.5,-0.8,0.3,9;
move 3,-523,0.5,-0.8,0.2,9;
move 2,-522.6,0.5,-0.8,0.1,9;
move 1,-522.2,0.5,-1.2,0,9;
move 0,-521.7,0.5,-1.2,-0.1,9;
move -1,-521.2,0.5,-1.2,-0.1,9;
move -2,-520.6,0.5,-1.2,-0.2,9;
move -3,-519.9,0.4,-1.2,-0.3,9;
move -4,-519.2,0.4,-1.2,-0.4,9;
move -5,-518.5,0.4,-1.2,-0.5,9;
move -5,-517.8,0.4,-1.6,-0.6,9;
move -6,-517,0.3,-1.6,-0.7,9;
move -7,-516.1,0.3,-1.6,-0.7,9;
move -7,-515.3,0.3,-1.6,-0.8,9;
move -8,-514.5,0.2,-1.6,-0.9,9;
move -8,-513.7,0.2,-1.6,-1,9;
move -8,-512.8,0.1,-1.6,-1.1,9;
move -9,-512,0.1,-1.6,-1.1,9;
move -9,-511.3,0,-1.6,-1.2,9;
move -10,-510.6,-0,-1.6,-1.3,9;
move -10,-509.9,-0.1,-1.6,-1.4,9;
move -11,-509.3,-0.1,-1.6,-1.5,9;
move -11,-508.7,-0.2,-2,-1.5,9;
move -12,-508.2,-0.2,-2,-1.6,9;
move -12,-507.8,-0.2,-2,-1.7,9;
move -13,-507.4,-0.3,-2,-1.8,9;
move -13,-507.1,-0.3,-2,-1.9,9;
move -13,-506.9,-0.4,-2,-1.9,9;
move -14,-506.8,-0.5,-2,-2,9;
move -14,-506.7,-0.5,-2,-2.1,9;
move -14,-506.6,-0.6,-2,-2.2,9;
move -14,-506.7,-0.7,-2,-2.2,9;
move -15,-506.8,-0.7,-2,-2.3,9;
move -15,-506.9,-0.8,-2,-2.4,8.9;
move -16,-507.1,-0.9,-2,-2.5,8.9;
move -16,-507.4,-0.9,-2,-2.5,8.9;
move -17,-507.7,-1,-2.4,-2.6,8.9;
move -17,-508.1,-1.1,-2.4,-2.7,8.9;
move -18,-508.5,-1.1,-2.4,-2.7,8.9;
move -18,-508.9,-1.2,-2.4,-2.8,8.9;
move -19,-509.4,-1.3,-2.4,-2.9,8.9;
move -19,-509.8,-1.4,-2.4,-2.9,8.9;
move -20,-510.3,-1.4,-2.4,-3,8.8;
move -20,-510.7,-1.5,-2.4,-3.1,8.8;
move -20,-511.2,-1.6,-2.4,-3.2,8.8;
move -21,-511.6,-1.6,-2.4,-3.2,8.8;
move -21,-512,-1.7,-2.4,-3.3,8.8;
move -22,-512.4,-1.8,-2.4,-3.4,8.7;
move -23,-512.7,-1.9,-2.8,-3.4,8.7;
move -23,-512.9,-1.9,-2.8,-3.5,8.7;
move -24,-513.1,-2,-2.8,-3.5,8.7;
move -24,-513.1,-2.1,-2.8,-3.6,8.7;
move -25,-513.1,-2.1,-2.8,-3.7,8.6;
move -25,-513,-2.2,-2.8,-3.7,8.6;
move -25,-512.8,-2.3,-2.8,-3.8,8.6;
move -26,-512.5,-2.3,-2.8,-3.9,8.5;
move -26,-512,-2.4,-2.8,-3.9,8.5;
move -26,-511.5,-2.5,-2.8,-4,8.5;
move -27,-510.9,-2.5,-2.8,-4,8.5;
move -27,-510.1,-2.6,-2.8,-4.1,8.4;
move -28,-509.3,-2.6,-3.2,-4.2,8.4;
move -28,-508.4,-2.7,-3.2,-4.2,8.4;
move -29,-507.3,-2.7,-3.2,-4.3,8.3;
move -29,-506.2,-2.7,-2.8,-4.3,8.3;
move -30,-505.1,-2.8,-3.2,-4.4,8.3;
move -30,-503.9,-2.8,-3.2,-4.4,8.2;
move -30,-502.6,-2.8,-3.2,-4.5,8.2;
move -30,-501.3,-2.9,-3.2,-4.6,8.2;
move -30,-500,-2.9,-3.2,-4.6,8.1;
move -30,-498.7,-3,-3.2,-4.7,8.1;
move -30,-497.4,-3,-3.2,-4.7,8.1;
move -30,-496.2,-3,-3.2,-4.8,8;
move -30,-495,-3,-3.2,-4.8,8;
move -29,-493.8,-3,-3.2,-4.9,8;
move -29,-492.6,-3,-3.2,-4.9,7.9;
move -28,-491.5,-3,-3.2,-5,7.9;
move -28,-490.5,-3,-2.8,-5,7.9;
move -27,-489.5,-3,-2.8,-5.1,7.8;
move -26,-488.6,-3,-2.8,-5.1,7.8;
move -26,-487.8,-3,-2.8,-5.2,7.8;
move -25,-487.1,-2.9,-2.8,-5.2,7.7;
move -25,-486.5,-2.9,-2.8,-5.3,7.7;
move -24,-486,-2.9,-2.8,-5.3,7.6;
move -23,-485.5,-2.9,-2.8,-5.4,7.6;
move -22,-485.1,-2.8,-2.8,-5.4,7.6;
move -21,-484.7,-2.8,-2.4,-5.5,7.5;
move -20,-484.5,-2.8,-2.4,-5.5,7.5;
move -19,-484.2,-2.7,-2.4,-5.5,7.5;
move -18,-484,-2.7,-2.4,-5.6,7.4;
move -17,-483.8,-2.7,-2.4,-5.6,7.4;
move -16,-483.7,-2.6,-2,-5.7,7.3;
move -15,-483.5,-2.6,-2,-5.7,7.3;
move -14,-483.4,-2.5,-2,-5.8,7.3;
move -13,-483.2,-2.5,-2,-5.8,7.2;
move -11,-483,-2.4,-2,-5.8,7.2;
move -10,-482.8,-2.4,-1.6,-5.9,7.1;
move -9,-482.6,-2.3,-1.6,-5.9,7.1;
move -8,-482.3,-2.3,-1.6,-6,7.1;
move -6,-482,-2.2,-1.6,-6,7;
move -5,-481.7,-2.1,-1.2,-6,7;
move -4,-481.5,-2,-1.2,-6.1,6.9;
move -3,-481.2,-2,-1.2,-6.1,6.9;
move -1,-480.8,-1.9,-1.2,-6.2,6.8;
move 0,-480.5,-1.8,-1.2,-6.2,6.8;
move 1,-480.2,-1.8,-0.8,-6.2,6.8;
move 2,-479.9,-1.7,-0.8,-6.3,6.7;
move 3,-479.7,-1.6,-0.8,-6.3,6.7;
move 4,-479.5,-1.5,-0.8,-6.3,6.6;
move 5,-479.3,-1.5,-0.8,-6.4,6.6;
move 7,-479.1,-1.4,-0.4,-6.4,6.5;
move 8,-479,-1.3,-0.4,-6.4,6.5;
move 9,-478.8,-1.2,-0.4,-6.5,6.5;
move 10,-478.8,-1.2,-0.4,-6.5,6.4;
move 11,-478.8,-1.1,-0.4,-6.5,6.4;
move 12,-478.8,-1,-0,-6.6,6.3;
move 13,-478.9,-1,-0,-6.6,6.3;
move 14,-479,-0.9,0,-6.6,6.2;
move 15,-479.2,-0.8,0,-6.7,6.2;
move 16,-479.4,-0.8,0,-6.7,6.1;
move 17,-479.6,-0.7,0,-6.7,6.1;
move 18,-479.8,-0.6,0.4,-6.7,6;
move 19,-480.1,-0.6,0.4,-6.8,6;
move 20,-480.4,-0.5,0.4,-6.8,5.9;
move 21,-480.8,-0.4,0.4,-6.8,5.9;
move 22,-481.2,-0.4,0.4,-6.9,5.8;
move 23,-481.6,-0.3,0.8,-6.9,5.8;
move 24,-482,-0.2,0.8,-6.9,5.8;
move 24,-482.4,-0.2,0.8,-6.9,5.7;
move 25,-482.9,-0.1,0.8,-7,5.7;
move 26,-483.3,-0,0.8,-7,5.6;
move 26,-483.7,0,0.8,-7,5.6;
move 27,-484.2,0.1,0.8,-7,5.5;
move 27,-484.6,0.2,0.8,-7.1,5.5;
move 28,-485,0.2,0.8,-7.1,5.4;
move 28,-485.5,0.3,0.8,-7.1,5.4;
move 29,-485.9,0.3,1.2,-7.1,5.3;
move 30,-486.3,0.4,1.2,-7.1,5.3;
move 30,-486.8,0.5,1.2,-7.2,5.2;
move 31,-487.2,0.5,1.2,-7.2,5.2;
move 31,-487.7,0.6,1.2,-7.2,5.1;
move 31,-488.2,0.6,1.2,-7.2,5.1;
move 31,-488.7,0.6,1.2,-7.3,5;
move 31,-489.2,0.7,1.2,-7.3,5;
move 32,-489.7,0.7,1.2,-7.3,4.9;
move 32,-490.2,0.7,1.2,-7.3,4.9;
move 32,-490.8,0.7,1.2,-7.3,4.8;
move 32,-491.3,0.8,1.2,-7.3,4.8;
move 32,-491.9,0.8,1.2,-7.4,4.7;
move 31,-492.4,0.9,1.2,-7.4,4.7;
move 31,-493,0.9,1.2,-7.4,4.6;
move 31,-493.5,1,1.2,-7.4,4.6;
move 31,-494,1,1.2,-7.4,4.5;
move 30,-494.5,1,1.2,-7.5,4.4;
move 30,-495,1,1.2,-7.5,4.4;
move 29,-495.4,1.1,1.2,-7.5,4.3;
move 28,-495.8,1.1,0.8,-7.5,4.3;
move 28,-496.1,1.1,0.8,-7.5,4.2;
move 27,-496.4,1.1,0.8,-7.5,4.2;
move 27,-496.7,1.1,0.8,-7.5,4.1;
move 26,-496.9,1.1,0.8,-7.6,4.1;
move 25,-497,1.1,0.8,-7.6,4;
move 25,-497.2,1.1,0.8,-7.6,4;
move 24,-497.2,1.2,0.8,-7.6,3.9;
move 23,-497.2,1.2,0.8,-7.6,3.9;
move 23,-497.2,1.2,0.4,-7.6,3.8;
move 22,-497.1,1.2,0.4,-7.6,3.7;
move 22,-497,1.2,0.4,-7.7,3.7;
move 21,-496.8,1.2,0.4,-7.7,3.6;
move 21,-496.5,1.2,0.4,-7.7,3.6;
move 20,-496.2,1.1,0.4,-7.7,3.5;
move 20,-495.9,1.1,0.4,-7.7,3.5;
move 19,-495.5,1.1,0.4,-7.7,3.4;
move 19,-495,1.1,0.4,-7.7,3.4;
move 18,-494.5,1,0.4,-7.7,3.3;
move 18,-494,1,0.4,-7.7,3.3;
move 17,-493.4,1,0,-7.8,3.2;
move 17,-492.8,0.9,0,-7.8,3.1;
move 16,-492.2,0.9,0,-7.8,3.1;
move 16,-491.6,0.9,0,-7.8,3;
move 15,-491,0.8,0,-7.8,3;
move 15,-490.4,0.8,-0,-7.8,2.9;
move 14,-489.8,0.7,-0,-7.8,2.9;
move 14,-489.3,0.7,-0,-7.8,2.8;
move 13,-488.8,0.6,-0,-7.8,2.8;
move 13,-488.3,0.6,-0,-7.8,2.7;
move 12,-487.9,0.5,-0,-7.8,2.6;
move 11,-487.5,0.5,-0.4,-7.9,2.6;
move 11,-487.3,0.4,-0.4,-7.9,2.5;
move 10,-487.1,0.4,-0.4,-7.9,2.5;
move 10,-487,0.3,-0.4,-7.9,2.4;
move 10,-486.9,0.2,-0.4,-7.9,2.4;
move 9,-487,0.2,-0.4,-7.9,2.3;
move 9,-487.1,0.1,-0.4,-7.9,2.3;
move 9,-487.3,0.1,-0.4,-7.9,2.2;
move 9,-487.5,-0,-0.4,-7.9,2.1;
move 9,-487.9,-0.1,-0.4,-7.9,2.1;
move 9,-488.3,-0.1,-0.4,-7.9,2;
move 9,-488.7,-0.2,-0.4,-7.9,2;
move 9,-489.2,-0.3,-0.4,-7.9,1.9;
move 9,-489.8,-0.3,-0.4,-7.9,1.9;
move 9,-490.3,-0.4,-0.4,-7.9,1.8;
move 9,-490.9,-0.5,-0.4,-8,1.8;
move 9,-491.5,-0.5,-0.4,-8,1.7;
move 9,-492,-0.6,-0.4,-8,1.6;
move 8,-492.6,-0.7,-0.4,-8,1.6;
move 8,-493.1,-0.7,-0.4,-8,1.5;
move 8,-493.6,-0.8,-0.4,-8,1.5;
move 8,-494.1,-0.8,-0.4,-8,1.4;
move 8,-494.5,-0.9,-0.8,-8,1.4;
move 8,-494.9,-1,-0.4,-8,1.3;
move 7,-495.2,-1,-0.4,-8,1.3;
move 7,-495.4,-1.1,-0.4,-8,1.2;
move 7,-495.6,-1.2,-0.8,-8,1.1;
move 8,-495.7,-1.2,-0.8,-8,1.1;
move 8,-495.8,-1.3,-0.4,-8,1;
move 8,-495.7,-1.3,-0.4,-8,1;
move 8,-495.7,-1.4,-0.4,-8,0.9;
move 8,-495.5,-1.4,-0.4,-8,0.9;
move 8,-495.3,-1.5,-0.4,-8,0.8;
move 9,-495,-1.5,-0.4,-8,0.8;
move 9,-494.7,-1.6,-0.4,-8,0.7;
move 9,-494.3,-1.6,-0.4,-8,0.6;
move 9,-493.9,-1.7,-0.4,-8,0.6;
move 9,-493.4,-1.7,-0.4,-8,0.5;
move 9,-492.8,-1.8,-0.4,-8,0.5;
move 9,-492.2,-1.8,-0.4,-8,0.4;
move 9,-491.6,-1.8,-0.4,-8,0.4;
move 9,-490.9,-1.9,-0.4,-8,0.3;
move 10,-490.2,-1.9,-0.4,-8,0.2;
move 10,-489.5,-1.9,-0.4,-8,0.2;
move 10,-488.8,-1.9,-0.4,-8,0.1;
move 11,-488,-2,-0.4,-8,0.1;
move 12,-487.3,-2,-0.4,-8,0;
move 12,-486.5,-2,-0,-8,-0;
move 13,-485.7,-2,-0,-8,-0.1;
move 14,-485,-2,-0,-8,-0.1;
move 15,-484.2,-2,0,-8,-0.2;
move 16,-483.5,-2.1,0,-8,-0.3;
move 17,-482.8,-2.1,0,-8,-0.3;
move 19,-482.1,-2.1,0.4,-8,-0.4;
move 20,-481.5,-2.1,0.4,-8,-0.4;
move 21,-480.9,-2.1,0.4,-8,-0.5;
move 22,-480.4,-2.1,0.4,-8,-0.5;
move 23,-479.9,-2.1,0.8,-8,-0.6;
move 25,-479.4,-2.1,0.8,-8,-0.7;
move 26,-479,-2.1,0.8,-8,-0.7;
move 27,-478.7,-2.1,0.8,-8,-0.8;
move 28,-478.4,-2.1,0.8,-8,-0.8;
move 29,-478.1,-2.1,1.2,-8,-0.9;
move 31,-477.9,-2.1,1.2,-8,-0.9;
move 32,-477.7,-2.1,1.2,-8,-1;
move 33,-477.6,-2.1,1.2,-8,-1.1;
move 34,-477.6,-2.1,1.2,-8,-1.1;
move 35,-477.6,-2.1,1.6,-8,-1.2;
move 37,-477.7,-2.1,1.6,-8,-1.2;
move 38,-477.8,-2,1.6,-8,-1.3;
move 39,-478,-2,1.6,-8,-1.3;
move 40,-478.3,-2,2,-8,-1.4;
move 41,-478.7,-2,2,-8,-1.5;
move 42,-479.1,-2,2,-8,-1.5;
move 43,-479.7,-2,2,-8,-1.6;
move 44,-480.3,-1.9,2,-8,-1.6;
move 45,-481,-1.9,2,-8,-1.7;
move 46,-481.8,-1.9,2.4,-8,-1.7;
move 47,-482.6,-1.9,2.4,-8,-1.8;
move 47,-483.6,-1.9,2.4,-8,-1.9;
move 48,-484.6,-1.8,2.4,-7.9,-1.9;
move 49,-485.7,-1.8,2.4,-7.9,-2;
move 49,-486.8,-1.8,2.4,-7.9,-2;
move 50,-488,-1.8,2.4,-7.9,-2.1;
move 51,-489.2,-1.8,2.4,-7.9,-2.1;
move 51,-490.4,-1.7,2.4,-7.9,-2.2;
move 52,-491.7,-1.7,2.8,-7.9,-2.2;
move 52,-492.9,-1.7,2.8,-7.9,-2.3;
move 53,-494.2,-1.7,2.8,-7.9,-2.4;
move 53,-495.4,-1.6,2.8,-7.9,-2.4;
move 53,-496.6,-1.6,2.8,-7.9,-2.5;
move 53,-497.8,-1.6,2.8,-7.9,-2.5;
move 53,-498.9,-1.5,2.8,-7.9,-2.6;
move 52,-500,-1.5,2.8,-7.9,-2.6;
move 52,-501,-1.4,2.8,-7.9,-2.7;
move 51,-501.9,-1.4,2.4,-7.8,-2.7;
move 50,-502.8,-1.4,2.4,-7.8,-2.8;
move 50,-503.6,-1.3,2.4,-7.8,-2.9;
move 49,-504.4,-1.3,2.4,-7.8,-2.9;
move 48,-505,-1.3,2.4,-7.8,-3;
move 48,-505.6,-1.3,2.4,-7.8,-3;
move 47,-506.1,-1.2,2.4,-7.8,-3.1;
move 46,-506.6,-1.2,2.4,-7.8,-3.1;
move 45,-507,-1.1,2,-7.8,-3.2;
move 44,-507.4,-1.1,2,-7.8,-3.2;
move 43,-507.7,-1,2,-7.8,-3.3;
move 42,-508,-1,2,-7.7,-3.3;
move 40,-508.2,-0.9,2,-7.7,-3.4;
move 39,-508.4,-0.9,1.6,-7.7,-3.5;
move 38,-508.5,-0.8,1.6,-7.7,-3.5;
move 36,-508.6,-0.8,1.6,-7.7,-3.6;
move 35,-508.7,-0.7,1.6,-7.7,-3.6;
move 33,-508.7,-0.7,1.2,-7.7,-3.7;
move 32,-508.7,-0.6,1.2,-7.7,-3.7;
move 30,-508.7,-0.6,1.2,-7.7,-3.8;
move 28,-508.7,-0.5,1.2,-7.6,-3.8;
move 27,-508.6,-0.5,0.8,-7.6,-3.9;
move 25,-508.6,-0.4,0.8,-7.6,-3.9;
move 23,-508.5,-0.4,0.4,-7.6,-4;
move 21,-508.5,-0.3,0.4,-7.6,-4;
move 18,-508.4,-0.2,0.4,-7.6,-4.1;
move 16,-508.4,-0.2,0,-7.6,-4.1;
move 14,-508.3,-0.1,-0,-7.5,-4.2;
move 12,-508.3,-0,-0,-7.5,-4.2;
move 9,-508.3,0,-0.4,-7.5,-4.3;
move 7,-508.2,0.1,-0.4,-7.5,-4.4;
move 4,-508.2,0.2,-0.8,-7.5,-4.4;
move 2,-508.2,0.2,-0.8,-7.5,-4.5;
move -1,-508.2,0.3,-1.2,-7.4,-4.5;
move -4,-508.1,0.4,-1.2,-7.4,-4.6;
move -7,-508.1,0.4,-1.6,-7.4,-4.6;
move -10,-508,0.5,-1.6,-7.4,-4.7;
move -13,-507.9,0.6,-2,-7.4,-4.7;
move -16,-507.8,0.7,-2,-7.4,-4.8;
move -19,-507.6,0.8,-2.4,-7.3,-4.8;
move -22,-507.4,0.9,-2.4,-7.3,-4.9;
move -25,-507.2,0.9,-2.8,-7.3,-4.9;
move -28,-506.9,1,-3.2,-7.3,-5;
move -31,-506.6,1.1,-3.2,-7.3,-5;
move -34,-506.2,1.2,-3.6,-7.2,-5.1;
move -37,-505.9,1.3,-3.6,-7.2,-5.1;
move -40,-505.5,1.4,-4,-7.2,-5.2;
move -42,-505.1,1.5,-4,-7.2,-5.2;
move -45,-504.7,1.6,-4,-7.2,-5.3;
move -48,-504.2,1.8,-4.4,-7.1,-5.3;
move -51,-503.8,1.9,-4.4,-7.1,-5.4;
move -54,-503.4,2,-4.8,-7.1,-5.4;
move -57,-503,2,-5.2,-7.1,-5.5;
move -60,-502.6,2.1,-5.2,-7,-5.5;
move -63,-502.2,2.2,-5.6,-7,-5.6;
move -66,-501.8,2.3,-5.6,-7,-5.6;
move -69,-501.4,2.4,-6,-7,-5.7;
move -72,-501,2.6,-6,-6.9,-5.7;
move -75,-500.6,2.7,-6.4,-6.9,-5.7;
move -78,-500.3,2.8,-6.4,-6.9,-5.8;
move -80,-499.9,2.9,-6.8,-6.9,-5.8;
move -83,-499.4,3,-6.8,-6.8,-5.9;
move -86,-499,3.1,-7.2,-6.8,-5.9;
move -89,-498.6,3.2,-7.2,-6.8,-6;
move -91,-498.2,3.3,-7.6,-6.8,-6;
move -94,-497.7,3.4,-7.6,-6.7,-6.1;
move -96,-497.2,3.5,-8,-6.7,-6.1;
move -99,-496.7,3.6,-8,-6.7,-6.2;
move -101,-496.1,3.7,-8,-6.6,-6.2;
move -103,-495.4,3.9,-8.4,-6.6,-6.3;
move -105,-494.7,4,-8.4,-6.6,-6.3;
move -107,-494,4.1,-8.8,-6.6,-6.4;
move -109,-493.2,4.2,-8.8,-6.5,-6.4;
move -111,-492.4,4.3,-8.8,-6.5,-6.5;
move -113,-491.4,4.4,-9.2,-6.5,-6.5;
move -115,-490.4,4.5,-9.2,-6.4,-6.5;
move -116,-489.4,4.6,-9.2,-6.4,-6.6;
move -117,-488.2,4.7,-9.2,-6.4,-6.6;
move -118,-487,4.8,-9.6,-6.3,-6.7;
move -119,-485.8,4.9,-9.6,-6.3,-6.7;
move -120,-484.4,5,-9.6,-6.3,-6.8;
move -121,-482.9,5.1,-9.6,-6.2,-6.8;
move -121,-481.4,5.2,-9.6,-6.2,-6.9;
move -121,-479.8,5.2,-9.6,-6.1,-6.9;
move -121,-478,5.3,-9.6,-6.1,-6.9;
move -122,-476.2,5.4,-9.6,-6.1,-7;
move -121,-474.2,5.5,-9.6,-6,-7;
move -121,-472.2,5.6,-9.6,-6,-7.1;
move -121,-470,5.7,-9.6,-6,-7.1;
move -120,-467.7,5.7,-9.6,-5.9,-7.2;
move -120,-465.2,5.8,-9.6,-5.9,-7.2;
move -119,-462.5,5.9,-9.6,-5.8,-7.2;
move -118,-459.8,6,-9.6,-5.8,-7.3;
move -116,-456.9,6.1,-9.2,-5.7,-7.3;
move -115,-453.9,6.1,-9.2,-5.7,-7.4;
move -113,-450.7,6.2,-9.2,-5.7,-7.4;
move -111,-447.4,6.2,-8.8,-5.6,-7.4;
move -109,-444,6.3,-8.8,-5.6,-7.5;
move -106,-440.6,6.3,-8.8,-5.5,-7.5;
move -103,-437.1,6.3,-8.4,-5.5,-7.5;
move -100,-433.6,6.4,-8,-5.4,-7.6;
move -97,-430.1,6.4,-8,-5.4,-7.6;
move -94,-426.6,6.4,-7.6,-5.4,-7.7;
move -91,-423.1,6.5,-7.6,-5.3,-7.7;
move -88,-419.6,6.5,-7.2,-5.3,-7.7;
move -84,-416.2,6.5,-6.8,-5.2,-7.8;
move -80,-412.9,6.5,-6.8,-5.2,-7.8;
move -77,-409.7,6.5,-6.4,-5.1,-7.8;
move -73,-406.7,6.5,-6.4,-5.1,-7.9;
move -69,-403.9,6.5,-6,-5,-7.9;
move -65,-401.3,6.5,-5.6,-5,-7.9;
move -61,-399,6.5,-5.2,-4.9,-8;
move -56,-396.9,6.5,-5.2,-4.9,-8;
move -52,-395,6.5,-4.8,-4.8,-8;
move -47,-393.5,6.4,-4.4,-4.8,-8.1;
move -43,-392.3,6.4,-4,-4.7,-8.1;
move -38,-391.5,6.4,-3.6,-4.6,-8.1;
move -33,-390.9,6.3,-3.2,-4.6,-8.2;
move -29,-390.8,6.3,-3.2,-4.5,-8.2;
move -24,-390.9,6.2,-2.8,-4.5,-8.2;
move -19,-391.5,6.2,-2.4,-4.4,-8.3;
move -15,-392.3,6.1,-2,-4.4,-8.3;
move -10,-393.4,6.1,-1.6,-4.3,-8.3;
move -6,-394.8,6,-1.2,-4.3,-8.4;
move -1,-396.5,6,-1.2,-4.2,-8.4;
move 3,-398.4,5.9,-0.8,-4.1,-8.4;
move 7,-400.5,5.8,-0.4,-4.1,-8.5;
move 11,-402.8,5.7,-0,-4,-8.5;
move 15,-405.3,5.6,0,-4,-8.5;
move 19,-407.8,5.6,0.4,-3.9,-8.5;
move 23,-410.5,5.5,0.8,-3.8,-8.6;
move 26,-413.3,5.4,0.8,-3.8,-8.6;
move 30,-416.1,5.3,1.2,-3.7,-8.6;
move 33,-418.9,5.2,1.2,-3.7,-8.7;
move 36,-421.7,5.1,1.6,-3.6,-8.7;
move 39,-424.5,5,2,-3.5,-8.7;
move 42,-427.3,4.9,2,-3.5,-8.7;
move 45,-430,4.8,2.4,-3.4,-8.7;
move 48,-432.7,4.7,2.4,-3.3,-8.8;
move 50,-435.2,4.6,2.4,-3.3,-8.8;
move 52,-437.8,4.5,2.8,-3.2,-8.8;
move 54,-440.2,4.4,2.8,-3.1,-8.8;
move 56,-442.5,4.3,3.2,-3.1,-8.8;
move 58,-444.6,4.2,3.2,-3,-8.9;
move 60,-446.7,4,3.2,-2.9,-8.9;
move 61,-448.6,3.9,3.2,-2.9,-8.9;
move 62,-450.4,3.8,3.6,-2.8,-8.9;
move 63,-452,3.7,3.6,-2.7,-8.9;
move 64,-453.4,3.6,3.6,-2.6,-8.9;
move 64,-454.8,3.4,3.6,-2.6,-8.9;
move 64,-456,3.3,3.6,-2.5,-8.9;
move 64,-457,3.2,3.6,-2.4,-8.9;
move 64,-458,3.1,3.6,-2.4,-8.9;
move 63,-458.8,3,3.6,-2.3,-9;
move 62,-459.5,2.9,3.6,-2.2,-9;
move 61,-460.2,2.8,3.2,-2.1,-9;
move 60,-460.8,2.7,3.2,-2.1,-9;
move 59,-461.2,2.6,3.2,-2,-9;
move 57,-461.6,2.5,3.2,-1.9,-9;
move 56,-461.9,2.4,2.8,-1.8,-9;
move 54,-462.2,2.3,2.8,-1.8,-9;
move 52,-462.4,2.2,2.8,-1.7,-9;
move 50,-462.6,2.1,2.4,-1.6,-9;
move 48,-462.8,2,2.4,-1.5,-9;
move 46,-462.9,1.9,2.4,-1.4,-9;
move 44,-463,1.8,2,-1.4,-9;
move 42,-463,1.8,2,-1.3,-9;
move 39,-463.1,1.7,1.6,-1.2,-9;
move 37,-463.1,1.6,1.6,-1.1,-9;
move 35,-463.1,1.5,1.6,-1,-9;
move 32,-463.1,1.4,1.2,-1,-9;
move 29,-463.1,1.4,1.2,-0.9,-9;
move 27,-463.1,1.3,0.8,-0.8,-9;
move 24,-463.1,1.2,0.8,-0.7,-9;
move 21,-463.1,1.1,0.4,-0.6,-9;
move 18,-463.1,1,0.4,-0.5,-9;
move 14,-463,0.9,0,-0.5,-9;
move 11,-463,0.9,-0.4,-0.4,-9;
move 8,-462.9,0.8,-0.4,-0.3,-9;
move 4,-462.8,0.7,-0.8,-0.2,-9;
move 1,-462.7,0.7,-0.8,-0.1,-9;
move -3,-462.6,0.6,-1.2,-0,-9;
move -7,-462.4,0.6,-1.6,0.1,-9;
move -10,-462.2,0.5,-1.6,0.1,-9;
move -14,-462,0.4,-2,0.2,-9;
move -18,-461.7,0.4,-2.4,0.3,-9;
move -22,-461.4,0.4,-2.4,0.4,-9;
move -26,-461.1,0.3,-2.8,0.5,-9;
move -30,-460.7,0.3,-3.2,0.6,-9;
move -34,-460.3,0.2,-3.6,0.7,-9;
move -39,-459.8,0.2,-3.6,0.8,-9;
move -43,-459.3,0.1,-4,0.8,-9;
move -47,-458.7,0.1,-4.4,0.9,-9;
move -51,-458.2,0,-4.8,1,-9;
move -55,-457.6,-0,-4.8,1.1,-9;
move -59,-457,-0.1,-5.2,1.2,-9;
move -63,-456.3,-0.1,-5.6,1.3,-9;
move -67,-455.7,-0.2,-6,1.4,-9;
move -71,-455.1,-0.2,-6,1.5,-9;
move -75,-454.5,-0.3,-6.4,1.6,-9;
move -78,-453.9,-0.3,-6.4,1.7,-9;
move -82,-453.2,-0.3,-6.8,1.8,-9;
move -85,-452.6,-0.3,-7.2,1.9,-8.9;
move -89,-452.1,-0.3,-7.2,1.9,-8.9;
move -92,-451.5,-0.3,-7.6,2,-8.9;
move -96,-450.9,-0.4,-7.6,2.1,-8.9;
move -99,-450.4,-0.4,-8,2.2,-8.9;
move -103,-449.8,-0.4,-8.4,2.3,-8.9;
move -106,-449.3,-0.5,-8.8,2.4,-8.9;
move -109,-448.7,-0.5,-8.8,2.5,-8.9;
move -113,-448.2,-0.5,-8.8,2.6,-8.9;
move -116,-447.5,-0.5,-9.2,2.7,-8.8;
move -119,-446.9,-0.6,-9.2,2.8,-8.8;
move -122,-446.1,-0.6,-9.6,2.9,-8.8;
move -126,-445.3,-0.6,-10,3,-8.8;
move -129,-444.3,-0.6,-10,3.1,-8.8;
move -132,-443.3,-0.6,-10.4,3.2,-8.7;
move -135,-442.1,-0.7,-10.8,3.3,-8.7;
move -138,-440.7,-0.7,-10.8,3.4,-8.7;
move -141,-439.3,-0.7,-11.2,3.5,-8.7;
move -143,-437.6,-0.7,-11.2,3.6,-8.6;
move -146,-435.8,-0.8,-11.6,3.7,-8.6;
move -148,-433.9,-0.8,-11.6,3.8,-8.6;
move -150,-431.8,-0.8,-11.6,3.9,-8.6;
move -152,-429.5,-0.8,-11.6,3.9,-8.5;
move -154,-427.2,-0.8,-11.6,4,-8.5;
move -156,-424.8,-0.8,-12,4.1,-8.5;
move -158,-422.2,-0.8,-12,4.2,-8.4;
move -159,-419.6,-0.8,-12.4,4.3,-8.4;
move -161,-417,-0.8,-12.4,4.4,-8.4;
move -162,-414.3,-0.8,-12.8,4.5,-8.3;
move -164,-411.5,-0.8,-12.8,4.6,-8.3;
move -165,-408.8,-0.9,-12.8,4.7,-8.3;
move -165,-406.1,-0.9,-12.8,4.8,-8.2;
move -166,-403.5,-0.9,-12.8,4.9,-8.2;
move -166,-400.9,-0.9,-12.8,5,-8.1;
move -166,-398.3,-0.9,-12.8,5.1,-8.1;
move -166,-395.8,-0.9,-12.8,5.2,-8.1;
move -166,-393.4,-0.9,-12.8,5.3,-8;
move -165,-391,-0.9,-12.8,5.4,-8;
move -165,-388.6,-0.9,-12.8,5.5,-7.9;
move -164,-386.3,-0.8,-12.4,5.6,-7.9;
move -163,-384,-0.8,-12.4,5.7,-7.9;
move -162,-381.7,-0.8,-12.4,5.8,-7.8;
move -162,-379.4,-0.8,-12.4,5.9,-7.8;
move -161,-377.2,-0.8,-12.4,6,-7.7;
move -160,-374.9,-0.8,-12.4,6.1,-7.7;
move -159,-372.5,-0.8,-12.4,6.2,-7.6;
move -158,-370.2,-0.8,-12,6.3,-7.6;
move -157,-367.7,-0.8,-12,6.4,-7.5;
move -156,-365.3,-0.8,-12,6.5,-7.5;
move -155,-362.9,-0.8,-12,6.5,-7.4;
move -154,-360.6,-0.8,-12,6.6,-7.4;
move -152,-358.1,-0.8,-12,6.7,-7.3;
move -151,-355.7,-0.8,-11.6,6.8,-7.3;
move -149,-353.3,-0.8,-11.6,6.9,-7.2;
move -147,-351,-0.8,-11.6,7,-7.2;
move -145,-348.6,-0.8,-11.2,7.1,-7.1;
move -142,-346.4,-0.8,-11.2,7.2,-7.1;
move -140,-344.2,-0.8,-10.8,7.3,-7;
move -137,-342.2,-0.8,-10.8,7.4,-7;
move -134,-340.4,-0.8,-10.4,7.5,-6.9;
move -132,-338.8,-0.8,-10.4,7.6,-6.9;
move -129,-337.5,-0.8,-10,7.7,-6.8;
move -126,-336.4,-0.8,-10,7.8,-6.7;
move -123,-335.6,-0.8,-9.6,7.9,-6.7;
move -121,-335,-0.8,-9.6,7.9,-6.6;
move -118,-334.8,-0.8,-9.2,8,-6.6;
move -115,-334.7,-0.8,-9.2,8.1,-6.5;
move -113,-334.9,-0.8,-8.8,8.2,-6.5;
move -110,-335.3,-0.9,-8.8,8.3,-6.4;
move -108,-336,-0.9,-8.4,8.4,-6.3;
move -105,-336.8,-0.9,-8.4,8.5,-6.3;
move -103,-337.8,-0.9,-8.4,8.6,-6.2;
move -101,-339,-1,-8,8.7,-6.1;
move -99,-340.3,-1,-8,8.7,-6.1;
move -97,-341.6,-1,-7.6,8.8,-6;
move -95,-343,-1,-7.6,8.9,-5.9;
move -94,-344.3,-1.1,-7.6,9,-5.9;
move -92,-345.5,-1.1,-7.6,9.1,-5.8;
move -91,-346.5,-1.1,-7.2,9.2,-5.7;
move -89,-347.3,-1.1,-7.2,9.3,-5.7;
move -88,-347.9,-1.2,-7.2,9.3,-5.6;
move -87,-348.2,-1.2,-7.2,9.4,-5.5;
move -86,-348.4,-1.2,-7.2,9.5,-5.5;
move -85,-348.3,-1.3,-6.8,9.6,-5.4;
move -85,-348.1,-1.3,-6.8,9.7,-5.3;
move -85,-347.7,-1.4,-6.8,9.7,-5.3;
move -85,-347.2,-1.4,-6.8,9.8,-5.2;
move -85,-346.4,-1.4,-6.8,9.9,-5.1;
move -85,-345.6,-1.5,-6.8,10,-5;
move -85,-344.6,-1.5,-7.2,10.1,-5;
move -86,-343.5,-1.6,-7.2,10.1,-4.9;
move -86,-342.4,-1.6,-7.2,10.2,-4.8;
move -87,-341.3,-1.6,-7.2,10.3,-4.7;
move -87,-340.1,-1.7,-7.2,10.4,-4.7;
move -87,-339,-1.7,-7.2,10.4,-4.6;
move -88,-338,-1.8,-7.2,10.5,-4.5;
move -88,-337,-1.8,-7.2,10.6,-4.4;
move -89,-336.1,-1.8,-7.2,10.7,-4.4;
move -89,-335.3,-1.9,-7.2,10.7,-4.3;
move -90,-334.4,-1.9,-7.2,10.8,-4.2;
move -91,-333.6,-2,-7.2,10.9,-4.1;
move -92,-333,-2,-7.6,10.9,-4;
move -93,-332.3,-2.1,-7.6,11,-4;
move -94,-331.8,-2.1,-7.6,11.1,-3.9;
move -96,-331.2,-2.2,-7.6,11.2,-3.8;
move -97,-330.7,-2.2,-8,11.2,-3.7;
move -99,-330.2,-2.3,-8,11.3,-3.6;
move -100,-329.7,-2.3,-8,11.4,-3.5;
move -102,-329.1,-2.4,-8,11.4,-3.5;
move -104,-328.5,-2.5,-8,11.5,-3.4;
move -107,-327.8,-2.5,-8.4,11.5,-3.3;
move -109,-327,-2.6,-8.8,11.6,-3.2;
move -112,-326.1,-2.7,-8.8,11.7,-3.1;
move -115,-325,-2.7,-9.2,11.7,-3;
move -118,-323.8,-2.8,-9.2,11.8,-3;
move -121,-322.6,-2.9,-9.6,11.8,-2.9;
move -124,-321.2,-2.9,-9.6,11.9,-2.8;
move -127,-319.8,-3,-10,12,-2.7;
move -130,-318.3,-3.1,-10,12,-2.6;
move -134,-316.8,-3.2,-10.4,12.1,-2.5;
move -137,-315.3,-3.2,-10.8,12.1,-2.4;
move -141,-313.8,-3.3,-10.8,12.2,-2.3;
move -144,-312.3,-3.3,-11.2,12.2,-2.3;
move -147,-311,-3.4,-11.6,12.3,-2.2;
move -150,-309.7,-3.5,-12,12.3,-2.1;
move -153,-308.6,-3.6,-12,12.4,-2;
move -156,-307.8,-3.6,-12,12.4,-1.9;
move -159,-307.2,-3.7,-12.4,12.5,-1.8;
move -162,-306.9,-3.7,-12.4,12.5,-1.7;
move -164,-306.6,-3.8,-12.4,12.6,-1.6;
move -167,-306.5,-3.8,-12.8,12.6,-1.5;
move -170,-306.4,-3.9,-12.8,12.6,-1.4;
move -172,-306.2,-4,-13.2,12.7,-1.3;
move -175,-306.1,-4,-13.2,12.7,-1.3;
move -178,-305.9,-4.1,-13.6,12.8,-1.2;
move -180,-305.6,-4.1,-14,12.8,-1.1;
move -183,-305,-4.2,-14,12.8,-1;
move -186,-304.1,-4.2,-14,12.9,-0.9;
move -188,-302.9,-4.3,-14.4,12.9,-0.8;
move -190,-301.2,-4.3,-14.4,13,-0.7;
move -192,-299,-4.4,-14.8,13,-0.6;
move -194,-296.3,-4.4,-14.8,13,-0.5;
move -196,-293,-4.4,-14.8,13,-0.4;
move -197,-289.1,-4.4,-15.2,13.1,-0.3;
move -199,-284.6,-4.4,-15.2,13.1,-0.2;
move -200,-279.5,-4.5,-15.2,13.1,-0.1;
move -201,-273.8,-4.5,-15.2,13.2,-0;
move -202,-267.5,-4.5,-15.2,13.2,0.1;
move -203,-260.7,-4.5,-15.2,13.2,0.2;
move -203,-253.3,-4.5,-15.6,13.2,0.3;
move -203,-245.4,-4.5,-15.2,13.3,0.4;
move -203,-237.1,-4.5,-15.6,13.3,0.5;
move -203,-228.4,-4.5,-15.6,13.3,0.6;
move -203,-219.4,-4.5,-15.6,13.3,0.7;
move -202,-210.2,-4.4,-15.6,13.3,0.8;
move -201,-200.8,-4.4,-15.2,13.3,0.9;
move -199,-191.5,-4.3,-15.2,13.4,1;
move -198,-182.3,-4.3,-14.8,13.4,1.1;
move -196,-173.2,-4.2,-14.8,13.4,1.2;
move -194,-164.4,-4.2,-14.8,13.4,1.3;
move -191,-155.9,-4.1,-14.8,13.4,1.3;
move -189,-147.8,-4,-14.4,13.4,1.4;
move -186,-140.2,-4,-14.4,13.4,1.5;
move -183,-133.1,-3.9,-14,13.4,1.6;
move -180,-126.6,-3.8,-13.6,13.4,1.7;
move -177,-120.8,-3.7,-13.6,13.4,1.8;
move -174,-115.6,-3.6,-13.2,13.4,1.9;
move -170,-111.1,-3.6,-12.8,13.4,2;
move -167,-107.4,-3.5,-12.8,13.4,2.1;
move -163,-104.3,-3.4,-12.4,13.4,2.2;
move -160,-101.9,-3.3,-12.4,13.4,2.3;
move -156,-100.2,-3.2,-12.4,13.4,2.4;
move -152,-99,-3.1,-12,13.4,2.5;
move -148,-98.4,-3,-11.6,13.4,2.6;
move -143,-98.2,-3,-11.2,13.4,2.7;
move -139,-98.6,-2.9,-10.8,13.4,2.8;
move -134,-99.3,-2.8,-10.4,13.4,2.9;
move -129,-100.4,-2.7,-10,13.4,3;
move -125,-101.7,-2.6,-9.6,13.4,3.1;
move -120,-103.4,-2.6,-9.2,13.4,3.2;
move -116,-105.1,-2.4,-9.2,13.3,3.3;
move -112,-107,-2.4,-8.8,13.3,3.4;
move -108,-108.9,-2.3,-8.4,13.3,3.5;
move -104,-110.6,-2.2,-8.4,13.3,3.6;
move -100,-112.2,-2.1,-8,13.3,3.7;
move -96,-113.5,-2,-8,13.3,3.8;
move -92,-114.7,-1.9,-7.6,13.2,3.9;
move -88,-115.6,-1.9,-7.2,13.2,4;
move -83,-116.4,-1.8,-6.8,13.2,4.1;
move -79,-116.9,-1.7,-6.8,13.2,4.2;
move -74,-117.1,-1.7,-6.4,13.1,4.3;
move -69,-117.1,-1.6,-6,13.1,4.4;
move -65,-116.9,-1.5,-5.6,13.1,4.5;
move -60,-116.5,-1.4,-5.2,13,4.6;
move -55,-115.9,-1.4,-4.8,13,4.7;
move -50,-115.2,-1.3,-4.4,13,4.7;
move -46,-114.4,-1.3,-4,12.9,4.8;
move -41,-113.6,-1.2,-4,12.9,4.9;
move -37,-112.9,-1.2,-3.6,12.9,5;
move -33,-112.2,-1.1,-3.2,12.8,5.1;
move -29,-111.4,-1.1,-2.8,12.8,5.2;
move -25,-110.7,-1,-2.8,12.7,5.3;
move -21,-110.1,-1,-2.4,12.7,5.4;
move -17,-109.5,-1,-2,12.6,5.5;
move -14,-108.9,-0.9,-2,12.6,5.6;
move -11,-108.4,-0.9,-1.6,12.6,5.7;
move -7,-107.9,-0.9,-1.6,12.5,5.8;
move -4,-107.5,-0.8,-1.2,12.5,5.9;
move -1,-107.2,-0.8,-1.2,12.4,5.9;
move 2,-107,-0.8,-0.8,12.3,6;
move 5,-106.8,-0.8,-0.8,12.3,6.1;
move 8,-106.8,-0.8,-0.4,12.2,6.2;
move 11,-106.9,-0.8,-0.4,12.2,6.3;
move 14,-107.1,-0.8,-0,12.1,6.4;
move 17,-107.4,-0.8,0,12.1,6.5;
move 20,-107.7,-0.8,0.4,12,6.6;
move 23,-108.1,-0.8,0.8,11.9,6.6;
move 26,-108.6,-0.8,0.8,11.9,6.7;
move 29,-109.2,-0.8,1.2,11.8,6.8;
move 32,-109.9,-0.8,1.2,11.8,6.9;
move 35,-110.6,-0.8,1.6,11.7,7;
move 38,-111.3,-0.8,1.6,11.6,7.1;
move 41,-112.1,-0.8,2,11.6,7.1;
move 44,-112.9,-0.8,2,11.5,7.2;
move 47,-113.8,-0.9,2.4,11.4,7.3;
move 50,-114.7,-0.9,2.4,11.3,7.4;
move 52,-115.6,-0.9,2.8,11.3,7.5;
move 55,-116.5,-0.9,2.8,11.2,7.6;
move 57,-117.4,-1,3.2,11.1,7.6;
move 59,-118.3,-1,3.2,11,7.7;
move 62,-119.2,-1,3.6,11,7.8;
move 64,-120.1,-1.1,3.6,10.9,7.9;
move 66,-121,-1.1,3.6,10.8,7.9;
move 67,-122,-1.2,3.6,10.7,8;
move 69,-122.9,-1.2,3.6,10.6,8.1;
move 71,-123.8,-1.3,4,10.6,8.2;
move 73,-124.7,-1.3,4,10.5,8.3;
move 75,-125.6,-1.4,4.4,10.4,8.3;
move 77,-126.5,-1.4,4.4,10.3,8.4;
move 79,-127.3,-1.5,4.8,10.2,8.5;
move 81,-128.1,-1.5,4.8,10.1,8.6;
move 83,-128.9,-1.6,4.8,10,8.6;
move 85,-129.6,-1.7,4.8,9.9,8.7;
move 87,-130.4,-1.7,5.2,9.8,8.8;
move 89,-131.2,-1.8,5.2,9.7,8.8;
move 90,-132,-1.9,5.2,9.7,8.9;
move 92,-132.7,-2,5.6,9.6,9;
move 94,-133.4,-2,5.6,9.5,9;
move 96,-134.1,-2.1,5.6,9.4,9.1;
move 97,-134.7,-2.1,6,9.3,9.2;
move 99,-135.3,-2.2,6,9.2,9.2;
move 100,-135.9,-2.3,6,9.1,9.3;
move 102,-136.5,-2.3,6.4,9,9.4;
move 103,-137,-2.4,6.4,8.9,9.4;
move 104,-137.5,-2.4,6.4,8.7,9.5;
move 106,-138,-2.5,6.4,8.6,9.6;
move 107,-138.5,-2.6,6.4,8.5,9.6;
move 108,-138.8,-2.6,6.4,8.4,9.7;
move 109,-139.2,-2.7,6.4,8.3,9.8;
move 111,-139.6,-2.7,6.8,8.2,9.8;
move 112,-140.1,-2.7,6.8,8.1,9.9;
move 114,-140.6,-2.8,7.2,8,9.9;
move 116,-141.2,-2.9,7.2,7.9,10;
move 117,-141.9,-2.9,7.2,7.8,10;
move 119,-142.5,-3,7.2,7.7,10.1;
move 121,-143.3,-3.1,7.6,7.5,10.2;
move 122,-144.2,-3.1,7.6,7.4,10.2;
move 124,-145.1,-3.2,7.6,7.3,10.3;
move 126,-146.2,-3.3,7.6,7.2,10.3;
move 127,-147.3,-3.3,8,7.1,10.4;
move 129,-148.5,-3.4,8,7,10.4;
move 130,-149.7,-3.5,8.4,6.8,10.5;
move 132,-151,-3.5,8.4,6.7,10.5;
move 133,-152.4,-3.6,8.4,6.6,10.6;
move 134,-153.7,-3.7,8.8,6.5,10.6;
move 135,-155,-3.7,8.8,6.3,10.7;
move 136,-156.3,-3.8,8.4,6.2,10.7;
move 137,-157.6,-3.9,8.4,6.1,10.8;
move 137,-158.8,-4,8.8,6,10.8;
move 138,-160.1,-4.1,8.4,5.8,10.9;
move 139,-161.3,-4.1,8.4,5.7,10.9;
move 140,-162.5,-4.2,8.8,5.6,10.9;
move 141,-163.6,-4.3,8.8,5.5,11;
move 143,-164.6,-4.3,9.2,5.3,11;
move 144,-165.6,-4.4,9.2,5.2,11.1;
move 145,-166.7,-4.4,9.2,5.1,11.1;
move 146,-167.6,-4.5,9.2,5,11.2;
move 147,-168.5,-4.5,9.6,4.8,11.2;
move 148,-169.4,-4.6,9.6,4.7,11.2;
move 148,-170.2,-4.6,9.6,4.6,11.3;
move 149,-171,-4.7,9.6,4.4,11.3;
move 149,-171.8,-4.7,9.6,4.3,11.3;
move 148,-172.5,-4.8,9.6,4.2,11.4;
move 148,-173.2,-4.9,9.6,4,11.4;
move 147,-173.9,-4.9,9.2,3.9,11.5;
move 147,-174.7,-5,9.2,3.8,11.5;
move 146,-175.4,-5.1,9.2,3.6,11.5;
move 146,-176.2,-5.1,9.2,3.5,11.5;
move 145,-177.1,-5.2,8.8,3.3,11.6;
move 145,-178,-5.3,9.2,3.2,11.6;
move 144,-179,-5.3,9.2,3.1,11.6;
move 144,-180.1,-5.4,9.2,2.9,11.7;
move 143,-181.3,-5.5,9.2,2.8,11.7;
move 142,-182.6,-5.6,9.2,2.7,11.7;
move 141,-184,-5.6,9.2,2.5,11.7;
move 140,-185.5,-5.7,8.8,2.4,11.8;
move 139,-187.1,-5.8,8.8,2.2,11.8;
move 138,-189,-5.9,8.8,2.1,11.8;
move 136,-191,-5.9,8.4,2,11.8;
move 134,-193.2,-6,8.4,1.8,11.8;
move 132,-195.6,-6,8.4,1.7,11.9;
move 130,-198.1,-6.1,8.4,1.5,11.9;
move 128,-200.8,-6.2,8,1.4,11.9;
move 125,-203.7,-6.2,8,1.2,11.9;
move 122,-206.6,-6.3,7.6,1.1,11.9;
move 120,-209.7,-6.4,7.6,1,11.9;
move 117,-212.9,-6.4,7.2,0.8,11.9;
move 114,-216,-6.5,6.8,0.7,11.9;
move 110,-219.2,-6.5,6.8,0.5,11.9;
move 107,-222.4,-6.5,6.4,0.4,11.9;
move 103,-225.5,-6.6,6.4,0.2,11.9;
move 100,-228.5,-6.6,6,0.1,11.9;
move 96,-231.5,-6.6,6,-0,11.9;
move 92,-234.2,-6.6,5.6,-0.2,11.9;
move 88,-236.9,-6.7,5.2,-0.3,11.9;
move 83,-239.3,-6.7,5.2,-0.5,11.9;
move 79,-241.6,-6.8,4.8,-0.6,11.9;
move 74,-243.6,-6.8,4,-0.8,11.9;
move 70,-245.4,-6.8,3.6,-0.9,11.9;
move 65,-247,-6.9,3.2,-1.1,11.9;
move 61,-248.3,-6.9,3.2,-1.2,11.9;
move 56,-249.4,-7,2.8,-1.3,11.9;
move 52,-250.3,-7,2.8,-1.5,11.9;
move 48,-251,-7,2.4,-1.6,11.9;
move 44,-251.4,-7,2,-1.8,11.9;
move 40,-251.7,-7,1.6,-1.9,11.9;
move 35,-251.8,-7.1,1.6,-2.1,11.8;
move 31,-251.7,-7.1,1.2,-2.2,11.8;
move 27,-251.5,-7.1,0.8,-2.3,11.8;
move 22,-251.1,-7.1,0.8,-2.5,11.8;
move 17,-250.6,-7.1,0.4,-2.6,11.8;
move 13,-249.9,-7.2,-0,-2.8,11.7;
move 8,-249.1,-7.2,-0.8,-2.9,11.7;
move 3,-248.3,-7.3,-0.8,-3.1,11.7;
move -2,-247.3,-7.3,-1.2,-3.2,11.7;
move -7,-246.1,-7.3,-1.6,-3.3,11.6;
move -11,-244.7,-7.3,-2,-3.5,11.6;
move -16,-243.3,-7.3,-2.4,-3.6,11.6;
move -21,-241.7,-7.3,-2.4,-3.8,11.6;
move -25,-240,-7.4,-2.8,-3.9,11.5;
move -29,-238.2,-7.4,-3.2,-4.1,11.5;
move -34,-236.4,-7.4,-3.2,-4.2,11.5;
move -38,-234.4,-7.4,-3.6,-4.3,11.4;
move -42,-232.3,-7.4,-4,-4.5,11.4;
move -46,-230.2,-7.5,-4.4,-4.6,11.4;
move -50,-228,-7.5,-4.8,-4.8,11.3;
move -54,-225.6,-7.5,-5.2,-4.9,11.3;
move -58,-223.2,-7.5,-5.2,-5,11.2;
move -61,-220.6,-7.5,-5.6,-5.2,11.2;
move -64,-217.8,-7.5,-5.6,-5.3,11.2;
move -67,-215.1,-7.5,-5.6,-5.4,11.1;
move -70,-212.2,-7.5,-6,-5.6,11.1;
move -73,-209.4,-7.5,-6,-5.7,11;
move -76,-206.4,-7.4,-6.4,-5.8,11;
move -78,-203.5,-7.4,-6.8,-6,10.9;
move -81,-200.6,-7.4,-6.8,-6.1,10.9;
move -83,-197.6,-7.4,-6.8,-6.2,10.9;
move -85,-194.8,-7.4,-7.2,-6.4,10.8;
move -87,-192,-7.3,-7.2,-6.5,10.8;
move -89,-189.2,-7.3,-7.6,-6.6,10.7;
move -91,-186.6,-7.3,-7.6,-6.8,10.7;
move -92,-184,-7.3,-7.6,-6.9,10.6;
move -94,-181.6,-7.2,-7.6,-7,10.6;
move -95,-179.3,-7.2,-7.6,-7.2,10.5;
move -96,-177.3,-7.2,-8,-7.3,10.5;
move -97,-175.4,-7.1,-8,-7.4,10.4;
move -97,-173.7,-7.1,-8,-7.6,10.4;
move -98,-172.1,-7,-8,-7.7,10.3;
move -98,-170.4,-7,-8,-7.8,10.2;
move -98,-168.7,-7,-8,-7.9,10.2;
move -99,-166.8,-6.9,-8,-8.1,10.1;
move -98,-165,-6.9,-8,-8.2,10.1;
move -98,-163.1,-6.8,-8,-8.3,10;
move -98,-161.1,-6.7,-8,-8.4,10;
move -97,-158.9,-6.7,-8,-8.5,9.9;
move -97,-156.5,-6.6,-8,-8.7,9.8;
move -96,-154,-6.5,-8,-8.8,9.8;
move -95,-151.3,-6.4,-7.6,-8.9,9.7;
move -94,-148.5,-6.3,-7.6,-9,9.7;
move -93,-145.5,-6.3,-7.6,-9.1,9.6;
move -92,-142.5,-6.2,-7.6,-9.3,9.5;
move -91,-139.3,-6.1,-7.6,-9.4,9.5;
move -90,-136,-6,-7.2,-9.5,9.4;
move -89,-132.6,-5.9,-7.2,-9.6,9.3;
move -87,-129.3,-5.8,-7.2,-9.7,9.3;
move -86,-126,-5.6,-7.2,-9.8,9.2;
move -85,-122.9,-5.5,-7.2,-9.9,9.1;
move -83,-119.8,-5.4,-6.8,-10,9;
move -82,-116.9,-5.4,-6.8,-10.2,9;
move -80,-114.1,-5.3,-6.8,-10.3,8.9;
move -79,-111.5,-5.2,-6.4,-10.4,8.8;
move -77,-109,-5.1,-6.4,-10.5,8.8;
move -75,-106.9,-5,-6.4,-10.6,8.7;
move -73,-104.8,-4.8,-6.4,-10.7,8.6;
move -71,-103,-4.7,-6,-10.8,8.5;
move -69,-101.3,-4.6,-6,-10.9,8.4;
move -67,-99.8,-4.5,-5.6,-11,8.4;
move -65,-98.4,-4.3,-5.6,-11.1,8.3;
move -63,-97.2,-4.2,-5.6,-11.2,8.2;
move -61,-96.2,-4.1,-5.2,-11.3,8.1;
move -59,-95.3,-4,-5.2,-11.4,8.1;
move -56,-94.4,-3.8,-5.2,-11.5,8;
move -54,-93.6,-3.7,-4.8,-11.6,7.9;
move -52,-92.7,-3.5,-4.8,-11.7,7.8;
move -49,-91.8,-3.4,-4.4,-11.8,7.7;
move -47,-90.7,-3.2,-4.4,-11.9,7.6;
move -44,-89.5,-3.1,-4,-11.9,7.6;
move -41,-88.2,-3,-4,-12,7.5;
move -39,-86.6,-2.8,-3.6,-12.1,7.4;
move -36,-84.9,-2.7,-3.6,-12.2,7.3;
move -34,-83,-2.6,-3.2,-12.3,7.2;
move -32,-80.9,-2.4,-3.2,-12.4,7.1;
move -29,-78.5,-2.3,-3.2,-12.5,7;
move -27,-76,-2.2,-3.2,-12.5,7;
move -24,-73.4,-2.1,-2.8,-12.6,6.9;
move -22,-70.7,-1.9,-2.4,-12.7,6.8;
move -19,-67.9,-1.8,-2.4,-12.8,6.7;
move -17,-65.2,-1.7,-2,-12.9,6.6;
move -14,-62.5,-1.6,-2,-12.9,6.5;
move -12,-59.9,-1.4,-2,-13,6.4;
move -10,-57.5,-1.3,-1.6,-13.1,6.3;
move -7,-55.1,-1.2,-1.6,-13.1,6.2;
move -5,-52.7,-1.1,-1.2,-13.2,6.1;
move -3,-50.5,-1,-1.2,-13.3,6.1;
move 0,-48.3,-0.9,-1.2,-13.4,6;
move 2,-46.4,-0.8,-0.8,-13.4,5.9;
move 4,-44.6,-0.7,-0.8,-13.5,5.8;
move 7,-43,-0.6,-0.4,-13.5,5.7;
move 9,-41.7,-0.5,-0.4,-13.6,5.6;
move 11,-40.5,-0.4,-0.4,-13.7,5.5;
move 14,-39.5,-0.3,-0,-13.7,5.4;
move 16,-38.9,-0.2,0,-13.8,5.3;
move 19,-38.5,-0.2,0.4,-13.8,5.2;
move 21,-38.4,-0.1,0.4,-13.9,5.1;
move 23,-38.6,0,0.8,-14,5;
move 25,-38.9,0.1,0.8,-14,4.9;
move 27,-39.5,0.2,1.2,-14.1,4.8;
move 29,-40.5,0.3,1.2,-14.1,4.7;
move 31,-41.7,0.4,1.2,-14.2,4.6;
move 32,-43.2,0.4,1.2,-14.2,4.5;
move 33,-45.1,0.5,1.2,-14.3,4.4;
move 34,-47.3,0.6,1.6,-14.3,4.3;
move 35,-49.8,0.6,1.6,-14.3,4.2;
move 36,-52.7,0.7,1.6,-14.4,4.1;
move 37,-55.9,0.7,1.6,-14.4,4;
move 37,-59.4,0.8,1.6,-14.5,3.9;
move 38,-63.3,0.8,1.6,-14.5,3.8;
move 39,-67.4,0.8,1.6,-14.5,3.7;
move 39,-71.7,0.9,2,-14.6,3.6;
move 39,-76.1,0.9,2,-14.6,3.5;
move 40,-80.7,0.9,1.6,-14.6,3.4;
move 40,-85.3,1,1.6,-14.7,3.3;
move 41,-90,1,1.6,-14.7,3.2;
move 41,-94.8,1,2,-14.7,3.1;
move 41,-99.5,1,2,-14.8,3;
move 41,-104.2,1.1,2,-14.8,2.9;
move 41,-108.7,1.1,2,-14.8,2.8;
move 41,-113.1,1.2,2,-14.8,2.7;
move 40,-117.2,1.2,2,-14.9,2.6;
move 39,-121.1,1.2,2,-14.9,2.4;
move 38,-124.6,1.2,2,-14.9,2.3;
move 37,-127.8,1.2,1.6,-14.9,2.2;
move 36,-130.6,1.1,1.6,-14.9,2.1;
move 35,-133,1.2,1.2,-14.9,2;
move 33,-135,1.2,1.2,-14.9,1.9;
move 32,-136.6,1.2,0.8,-15,1.8;
move 31,-138,1.2,0.8,-15,1.7;
move 30,-139,1.2,1.2,-15,1.6;
move 28,-139.7,1.2,1.2,-15,1.5;
move 27,-140.1,1.2,1.2,-15,1.4;
move 26,-140.3,1.2,0.8,-15,1.3;
move 25,-140.2,1.2,0.8,-15,1.2;
move 23,-139.8,1.2,0.8,-15,1.1;
move 22,-139.3,1.2,0.4,-15,1;
move 20,-138.6,1.2,0.4,-15,0.9;
move 19,-137.7,1.2,0.4,-15,0.7;
move 17,-136.5,1.3,0,-15,0.6;
move 15,-135.2,1.3,-0,-15,0.5;
move 14,-133.7,1.3,-0,-15,0.4;
move 13,-132.1,1.3,-0.4,-15,0.3;
move 12,-130.4,1.4,-0.4,-15,0.2;
move 11,-128.5,1.4,-0.4,-14.9,0.1;
move 10,-126.5,1.4,-0.4,-14.9,0;
move 10,-124.5,1.5,-0.4,-14.9,-0.1;
move 9,-122.4,1.5,-0.4,-14.9,-0.2;
move 9,-120.2,1.5,-0.4,-14.9,-0.3;
move 9,-118,1.6,-0.4,-14.9,-0.4;
move 9,-115.7,1.6,-0.4,-14.9,-0.5;
move 10,-113.5,1.6,-0.4,-14.8,-0.6;
move 10,-111.2,1.6,-0.4,-14.8,-0.7;
move 10,-109,1.7,-0.4,-14.8,-0.8;
move 11,-106.8,1.7,-0.4,-14.8,-0.9;
move 11,-104.7,1.7,-0.4,-14.7,-1;
move 12,-102.7,1.8,-0,-14.7,-1.1;
move 13,-100.8,1.8,-0,-14.7,-1.3;
move 13,-99,1.8,0,-14.7,-1.4;
move 14,-97.3,1.9,0,-14.6,-1.5;
move 15,-95.8,1.9,0,-14.6,-1.6;
move 16,-94.4,1.9,0,-14.6,-1.7;
move 17,-93.1,1.9,-0,-14.5,-1.8;
move 18,-92.1,2,0,-14.5,-1.9;
move 19,-91.2,2,0,-14.4,-2;
move 21,-90.5,2,0.4,-14.4,-2.1;
move 22,-89.9,2.1,0.4,-14.4,-2.2;
move 24,-89.4,2.1,0.8,-14.3,-2.3;
move 26,-89.1,2.2,0.8,-14.3,-2.4;
move 29,-89,2.2,0.8,-14.2,-2.5;
move 31,-89.1,2.3,1.2,-14.2,-2.6;
move 33,-89.3,2.4,1.2,-14.1,-2.7;
move 36,-89.7,2.4,1.6,-14.1,-2.8;
move 38,-90.3,2.5,1.6,-14,-2.9;
move 41,-90.9,2.6,2,-14,-3;
move 43,-91.6,2.6,2,-13.9,-3.1;
move 45,-92.4,2.7,2,-13.9,-3.2;
move 48,-93.3,2.8,2.4,-13.8,-3.3;
move 51,-94.3,2.8,2.4,-13.8,-3.4;
move 53,-95.2,2.9,2.8,-13.7,-3.5;
move 56,-96.3,3,2.8,-13.7,-3.6;
move 59,-97.4,3.1,3.2,-13.6,-3.7;
move 62,-98.5,3.1,3.2,-13.5,-3.8;
move 65,-99.8,3.2,3.6,-13.5,-3.9;
move 68,-101,3.3,3.6,-13.4,-3.9;
move 70,-102.3,3.3,4,-13.4,-4;
move 73,-103.6,3.4,4.4,-13.3,-4.1;
move 76,-104.9,3.5,4.4,-13.2,-4.2;
move 78,-106.3,3.5,4.4,-13.2,-4.3;
move 81,-107.5,3.6,4.8,-13.1,-4.4;
move 84,-108.8,3.6,4.8,-13,-4.5;
move 86,-110,3.7,5.2,-13,-4.6;
move 88,-111.2,3.7,5.2,-12.9,-4.7;
move 91,-112.3,3.8,5.2,-12.8,-4.8;
move 93,-113.4,3.8,5.6,-12.7,-4.9;
move 96,-114.5,3.9,5.6,-12.7,-5;
move 98,-115.6,3.9,6,-12.6,-5;
move 101,-116.6,4,6,-12.5,-5.1;
move 103,-117.7,4,6.4,-12.4,-5.2;
move 105,-118.8,4.1,6.4,-12.4,-5.3;
move 108,-119.9,4.1,6.4,-12.3,-5.4;
move 111,-121.1,4.2,6.8,-12.2,-5.5;
move 113,-122.2,4.3,6.8,-12.1,-5.6;
move 116,-123.4,4.3,7.2,-12,-5.6;
move 118,-124.5,4.4,7.2,-11.9,-5.7;
move 121,-125.7,4.4,7.6,-11.9,-5.8;
move 124,-126.8,4.4,7.6,-11.8,-5.9;
move 126,-128,4.5,8,-11.7,-6;
move 129,-129.1,4.5,8,-11.6,-6.1;
move 131,-130.1,4.6,8.4,-11.5,-6.1;
move 133,-131.2,4.6,8.4,-11.4,-6.2;
move 135,-132.2,4.6,8.4,-11.3,-6.3;
move 138,-133.1,4.7,8.8,-11.2,-6.4;
move 140,-134,4.7,8.8,-11.2,-6.5;
move 141,-134.8,4.7,9.2,-11.1,-6.5;
move 143,-135.6,4.7,9.2,-11,-6.6;
move 145,-136.4,4.7,9.2,-10.9,-6.7;
move 146,-137.2,4.8,9.2,-10.8,-6.8;
move 148,-137.9,4.8,9.2,-10.7,-6.9;
move 150,-138.6,4.8,9.6,-10.6,-6.9;
move 151,-139.3,4.8,9.6,-10.5,-7;
move 153,-139.9,4.8,9.6,-10.4,-7.1;
move 154,-140.6,4.9,10,-10.3,-7.1;
move 156,-141.3,4.9,10,-10.2,-7.2;
move 157,-142,4.9,10,-10.1,-7.3;
move 158,-142.9,4.9,10.4,0,-7.4;
move 159,-143.7,4.9,10.4,0,-7.4;
move 160,-144.6,4.9,10.4,0,-7.5;
move 161,-145.5,4.9,10.4,0,-7.6;
move 162,-146.4,4.9,10.4,0,-7.6;
move 162,-147.5,4.9,10.4,0,-7.7;
move 163,-148.6,4.9,10.4,0,-7.8;
move 163,-149.8,4.9,10.4,0,-7.8;
move 164,-151,4.9,10.4,0,-7.9;
move 164,-152.4,4.8,10.4,0,-8;
move 164,-153.9,4.8,10.4,0,-8;
move 165,-155.5,4.8,10.8,0,-8.1;
move 165,-157.2,4.8,10.8,0,-8.1;
move 165,-159,4.8,10.8,0,-8.2;
move 165,-161,4.7,10.8,0,-8.3;
move 165,-163,4.7,10.8,0,-8.3;
move 164,-165.2,4.7,10.4,0,-8.4;
move 164,-167.4,4.7,10.4,0,-8.4;
move 163,-169.7,4.6,10.4,0,-8.5;
move 162,-172.1,4.6,10.4,0,-8.6;
move 161,-174.5,4.5,10.4,0,-8.6;
move 160,-176.9,4.5,10.4,0,-8.7;
move 159,-179.2,4.4,10.4,0,-8.7;
move 157,-181.6,4.4,10,-7.5,-8.8;
move 156,-184,4.3,10,-7.4,-8.8;
move 154,-186.3,4.2,10,-7.3,-8.9;
move 153,-188.6,4.2,9.6,-7.2,-8.9;
move 151,-190.8,4.2,9.6,-7.1,-9;
move 149,-192.9,4.1,9.6,-6.9,-9;
move 148,-195,4.1,9.2,-6.8,-9.1;
move 146,-197,4,9.2,-6.7,-9.1;
move 144,-198.9,3.9,9.2,-6.6,-9.2;
move 142,-200.7,3.9,9.2,-6.5,-9.2;
move 139,-202.5,3.8,8.8,-6.4,-9.2;
move 137,-204.1,3.8,8.8,-6.2,-9.3;
move 135,-205.6,3.7,8.4,-6.1,-9.3;
move 132,-207.1,3.6,8.4,-6,-9.4;
move 129,-208.5,3.6,8,-5.9,-9.4;
move 127,-209.8,3.5,8,-5.8,-9.4;
move 124,-210.9,3.4,7.6,-5.7,-9.5;
move 121,-212.1,3.4,7.6,-5.5,-9.5;
move 118,-213.1,3.3,7.2,-5.4,-9.6;
move 114,-214.1,3.2,7.2,-5.3,-9.6;
move 111,-215,3.1,6.8,-5.2,-9.6;
move 108,-215.9,3,6.4,-5.1,-9.6;
move 105,-216.8,2.9,6.4,-4.9,-9.7;
move 101,-217.7,2.8,6,-4.8,-9.7;
move 98,-218.5,2.7,6,-4.7,-9.7;
move 95,-219.4,2.7,5.6,-4.6,-9.7;
move 91,-220.2,2.6,5.6,-4.5,-9.8;
move 88,-221,2.5,5.2,-4.3,-9.8;
move 84,-221.9,2.4,4.8,-4.2,-9.8;
move 80,-222.8,2.3,4.8,-4.1,-9.8;
move 76,-223.6,2.3,4.4,-4,-9.8;
move 72,-224.5,2.2,4,-3.9,-9.9;
move 68,-225.3,2.1,3.6,-3.8,-9.9;
move 64,-226.2,2,3.6,-3.6,-9.9;
move 60,-227,1.9,3.2,-3.5,-9.9;
move 56,-227.8,1.8,2.8,-3.4,-9.9;
move 52,-228.5,1.7,2.4,-3.3,-9.9;
move 48,-229.2,1.6,2.4,-3.2,-9.9;
move 44,-229.9,1.5,2,-3,-9.9;
move 41,-230.5,1.4,1.6,-2.9,-9.9;
move 37,-231,1.3,1.6,-2.8,-10;
move 34,-231.5,1.2,1.2,-2.7,-10;
move 30,-231.8,1.1,1.2,-2.6,-10;
move 27,-232,1,0.8,-2.4,-10;
move 23,-232.1,0.9,0.8,-2.3,-10;
move 20,-232.1,0.8,0.4,-2.2,-10;
move 16,-231.9,0.7,0,-2.1,-10;
move 13,-231.6,0.6,-0,-2,-10;
move 10,-231.1,0.6,-0.4,-1.8,-10;
move 6,-230.6,0.5,-0.8,-1.7,-10;
move 3,-230,0.4,-0.8,-1.6,-10;
move 0,-229.2,0.3,-1.2,-1.5,-10;
move -3,-228.4,0.2,-1.2,-1.4,-10;
move -6,-227.4,0.2,-1.6,-1.3,-10;
move -9,-226.3,0.1,-1.6,-1.1,-10;
move -12,-225.1,0,-2,-1,-10;
move -14,-223.9,-0.1,-2,-0.9,-10;
move -17,-222.6,-0.1,-2.4,-0.8,-10;
move -19,-221.2,-0.2,-2.4,-0.7,-10;
move -21,-219.8,-0.2,-2.4,-0.6,-10;
move -24,-218.4,-0.3,-2.8,-0.4,-10;
move -26,-216.9,-0.3,-2.8,-0.3,-10;
move -28,-215.4,-0.4,-3.2,-0.2,-10;
move -30,-214,-0.4,-3.2,-0.1,-10;
move -32,-212.5,-0.5,-3.2,0,-10;
move -34,-211.1,-0.5,-3.6,0.1,-10;
move -36,-209.7,-0.6,-3.6,0.2,-10;
move -37,-208.3,-0.6,-3.6,0.3,-10;
move -39,-207,-0.7,-4,0.5,-10;
move -40,-205.8,-0.7,-4,0.6,-10;
move -42,-204.6,-0.8,-4,0.7,-10;
move -43,-203.5,-0.8,-4,0.8,-10;
move -44,-202.4,-0.8,-4,0.9,-10;
move -45,-201.4,-0.8,-4.4,1,-10;
move -46,-200.5,-0.9,-4.4,1.1,-10;
move -47,-199.7,-0.9,-4.4,1.2,-10;
move -47,-198.9,-0.9,-4.4,1.3,-10;
move -48,-198.2,-0.9,-4.4,1.4,-10;
move -48,-197.5,-0.9,-4.4,1.6,-10;
move -49,-196.8,-0.9,-4.4,1.7,-10;
move -49,-196.3,-0.9,-4.4,1.8,-10;
move -49,-195.8,-0.9,-4.4,1.9,-10;
move -50,-195.3,-0.9,-4.8,2,-10;
move -50,-194.8,-0.9,-4.8,2.1,-10;
move -50,-194.3,-0.9,-4.8,2.2,-10;
move -49,-193.9,-0.9,-4.4,2.3,-10;
move -49,-193.5,-0.9,-4.4,2.4,-10;
move -49,-193.1,-0.9,-4.4,2.5,-10;
move -49,-192.6,-0.9,-4.4,2.6,-9.9;
move -48,-192.2,-0.8,-4.4,2.7,-9.9;
move -48,-191.8,-0.8,-4.4,2.8,-9.9;
move -47,-191.4,-0.8,-4.4,2.9,-9.9;
move -47,-191,-0.7,-4.4,3,-9.9;
move -46,-190.6,-0.7,-4.4,3.1,-9.9;
move -46,-190.2,-0.7,-4.4,3.2,-9.9;
move -45,-189.8,-0.7,-4.4,3.3,-9.9;
move -44,-189.4,-0.6,-4,3.4,-9.9;
move -43,-188.9,-0.6,-4,3.5,-9.8;
move -41,-188.4,-0.5,-4,3.6,-9.8;
move -40,-187.9,-0.5,-4,3.7,-9.8;
move -39,-187.3,-0.4,-3.6,3.8,-9.8;
move -37,-186.8,-0.4,-3.6,3.9,-9.8;
move -36,-186.2,-0.3,-3.6,4,-9.7;
move -35,-185.6,-0.3,-3.6,4.1,-9.7;
move -33,-185,-0.2,-3.2,4.1,-9.7;
move -32,-184.4,-0.2,-3.2,4.2,-9.7;
move -31,-183.9,-0.1,-3.2,4.3,-9.6;
move -30,-183.3,-0.1,-3.2,4.4,-9.6;
move -28,-182.7,-0,-3.2,4.5,-9.6;
move -27,-182.1,0,-2.8,4.6,-9.5;
move -26,-181.5,0.1,-2.8,4.7,-9.5;
move -24,-181,0.1,-2.8,4.8,-9.5;
move -23,-180.4,0.2,-2.8,4.8,-9.4;
move -22,-179.9,0.2,-2.4,4.9,-9.4;
move -20,-179.5,0.3,-2.4,5,-9.4;
move -18,-179,0.3,-2.4,5.1,-9.3;
move -17,-178.6,0.4,-2.4,5.2,-9.3;
move -15,-178.2,0.5,-2,5.3,-9.3;
move -14,-177.9,0.5,-2,5.3,-9.2;
move -12,-177.6,0.6,-2,5.4,-9.2;
move -10,-177.3,0.6,-1.6,5.5,-9.1;
move -8,-177,0.7,-1.6,5.6,-9.1;
move -7,-176.8,0.7,-1.6,5.7,-9.1;
move -5,-176.6,0.8,-1.2,5.7,-9;
move -3,-176.4,0.9,-1.2,5.8,-9;
move -2,-176.3,0.9,-1.2,5.9,-8.9;
move 0,-176.2,1,-1.2,6,-8.9;
move 2,-176.1,1,-0.8,6,-8.8;
move 3,-176,1.1,-0.8,6.1,-8.8;
move 5,-175.9,1.1,-0.8,6.2,-8.8;
move 7,-175.8,1.2,-0.4,6.3,-8.7;
move 9,-175.8,1.2,-0.4,6.3,-8.7;
move 11,-175.8,1.2,-0.4,6.4,-8.6;
move 12,-175.8,1.3,-0,6.5,-8.6;
move 14,-175.8,1.3,0,6.5,-8.5;
move 16,-175.8,1.4,0,6.6,-8.5;
move 18,-175.9,1.4,0.4,6.7,-8.4;
move 19,-175.9,1.5,0.4,6.7,-8.4;
move 21,-175.9,1.5,0.4,6.8,-8.3;
move 23,-176,1.5,0.4,6.9,-8.3;
move 25,-176,1.6,0.8,6.9,-8.2;
move 26,-176,1.6,0.8,7,-8.2;
move 28,-176.1,1.6,0.8,7.1,-8.1;
move 30,-176.1,1.7,1.2,7.1,-8.1;
move 32,-176.1,1.7,1.2,7.2,-8;
move 33,-176.1,1.8,1.6,7.2,-7.9;
move 35,-176.1,1.8,1.6,7.3,-7.9;
move 36,-176.2,1.8,1.6,7.4,-7.8;
move 38,-176.2,1.9,1.6,7.4,-7.8;
move 39,-176.2,1.9,1.6,7.5,-7.7;
move 40,-176.2,1.9,1.6,7.5,-7.7;
move 42,-176.3,1.9,2,7.6,-7.6;
move 43,-176.4,1.9,2,7.6,-7.6;
move 44,-176.6,2,2,7.7,-7.5;
move 45,-176.7,2,2.4,7.7,-7.4;
move 47,-176.9,2,2.4,7.8,-7.4;
move 48,-177.2,2,2.4,7.8,-7.3;
move 49,-177.5,2,2.4,7.9,-7.3;
move 50,-177.8,1.9,2.4,7.9,-7.2;
move 51,-178.2,2,2.4,8,-7.2;
